LIN {X 0,Y 87.891,Z 1219.976,A -85,B 0,C 180,E1 32199.229,E2 32199.229} C_VEL
LIN {X 0,Y 83.761,Z 1226.847,A -85,B 0,C 180,E1 32206.195,E2 32206.195} C_VEL
LIN {X 0,Y 77.904,Z 1236.707,A -85,B 0,C 180,E1 32219.704,E2 32219.704} C_VEL
LIN {X 0,Y 80.765,Z 1249.005,A -85,B 0,C 180,E1 32238.354,E2 32238.354} C_VEL
LIN {X 0,Y 97.105,Z 1263.122,A -85,B 0,C 180,E1 32262.701,E2 32262.701} C_VEL
LIN {X 0,Y 95.268,Z 1262.7,A -85,B 0,C 180,E1 32265.572,E2 32265.572} C_VEL
LIN {X 0,Y 81.258,Z 1251.243,A -85,B 0,C 180,E1 32296.572,E2 32296.572} C_VEL
LIN {X 0,Y 81.376,Z 1245.78,A -85,B 0,C 180,E1 32307.381,E2 32307.381} C_VEL
LIN {X 0,Y 84.468,Z 1224.374,A -85,B 0,C 180,E1 32333.558,E2 32333.558} C_VEL
LIN {X 0,Y 99.54,Z 1230.344,A -85,B 0,C 180,E1 32359.626,E2 32359.626} C_VEL
LIN {X 0,Y 109.101,Z 1231.557,A -85,B 0,C 180,E1 32366.508,E2 32366.508} C_VEL
LIN {X 0,Y 89.421,Z 1216.791,A -85,B 0,C 180,E1 32382.617,E2 32382.617} C_VEL
LIN {X 0,Y 79.635,Z 1196.68,A -85,B 0,C 180,E1 32404.169,E2 32404.169} C_VEL
LIN {X 0,Y 80.434,Z 1173.933,A -85,B 0,C 180,E1 32423.679,E2 32423.679} C_VEL
LIN {X 0,Y 87.564,Z 1144.411,A -85,B 0,C 180,E1 32440.462,E2 32440.462} C_VEL
LIN {X 0,Y 96.99,Z 1111.48,A -85,B 0,C 180,E1 32451.459,E2 32451.459} C_VEL
LIN {X 0,Y 103.746,Z 1084.246,A -85,B 0,C 180,E1 32457.336,E2 32457.336} C_VEL
LIN {X 0,Y 98.146,Z 1049.051,A -85,B 0,C 180,E1 32468.442,E2 32468.442} C_VEL
LIN {X 0,Y 97.255,Z 1043.42,A -85,B 0,C 180,E1 32470.62,E2 32470.62} C_VEL
LIN {X 0,Y 108.101,Z 1031.914,A -85,B 0,C 180,E1 32479.137,E2 32479.137} C_VEL
LIN {X 0,Y 113.422,Z 1053.158,A -85,B 0,C 180,E1 32489.964,E2 32489.964} C_VEL
LIN {X 0,Y 118.845,Z 1081.531,A -85,B 0,C 180,E1 32501.191,E2 32501.191} C_VEL
LIN {X 0,Y 122.921,Z 1111.426,A -85,B 0,C 180,E1 32511.669,E2 32511.669} C_VEL
LIN {X 0,Y 123.967,Z 1124.968,A -85,B 0,C 180,E1 32516.233,E2 32516.233} C_VEL
LIN {X 0,Y 105.518,Z 1162.751,A -85,B 0,C 180,E1 32526.032,E2 32526.032} C_VEL
LIN {X 0,Y 89.617,Z 1194.356,A -85,B 0,C 180,E1 32540.566,E2 32540.566} C_VEL
LIN {X 0,Y 79.544,Z 1220.884,A -85,B 0,C 180,E1 32561.434,E2 32561.434} C_VEL
LIN {X 0,Y 77.904,Z 1236.707,A -85,B 0,C 180,E1 32579.704,E2 32579.704} C_VEL
LIN {X 0,Y 76.332,Z 1241.977,A -85,B 0,C 180,E1 32588.571,E2 32588.571} C_VEL
LIN {X 0,Y 75.282,Z 1248.971,A -85,B 0,C 180,E1 32604.581,E2 32604.581} C_VEL
LIN {X 0,Y 88.436,Z 1259.457,A -85,B 0,C 180,E1 32623.162,E2 32623.162} C_VEL
LIN {X 0,Y 74.447,Z 1249.413,A -85,B 0,C 180,E1 32652.297,E2 32652.297} C_VEL
LIN {X 0,Y 73.972,Z 1242.557,A -85,B 0,C 180,E1 32667.119,E2 32667.119} C_VEL
LIN {X 0,Y 77.694,Z 1220.967,A -85,B 0,C 180,E1 32695.202,E2 32695.202} C_VEL
LIN {X 0,Y 96.727,Z 1227.821,A -85,B 0,C 180,E1 32724.628,E2 32724.628} C_VEL
LIN {X 0,Y 98.246,Z 1227.61,A -85,B 0,C 180,E1 32726.965,E2 32726.965} C_VEL
LIN {X 0,Y 77.889,Z 1209.389,A -85,B 0,C 180,E1 32746.807,E2 32746.807} C_VEL
LIN {X 0,Y 71.41,Z 1187.367,A -85,B 0,C 180,E1 32770.787,E2 32770.787} C_VEL
LIN {X 0,Y 74.839,Z 1162.016,A -85,B 0,C 180,E1 32791.346,E2 32791.346} C_VEL
LIN {X 0,Y 83.559,Z 1131.844,A -85,B 0,C 180,E1 32806.599,E2 32806.599} C_VEL
LIN {X 0,Y 93.999,Z 1095.283,A -85,B 0,C 180,E1 32816.978,E2 32816.978} C_VEL
LIN {X 0,Y 96.451,Z 1084.975,A -85,B 0,C 180,E1 32819.249,E2 32819.249} C_VEL
LIN {X 0,Y 92.458,Z 1055.079,A -85,B 0,C 180,E1 32829.571,E2 32829.571} C_VEL
LIN {X 0,Y 102.072,Z 1044.415,A -85,B 0,C 180,E1 32837.324,E2 32837.324} C_VEL
LIN {X 0,Y 105.365,Z 1042.471,A -85,B 0,C 180,E1 32840.02,E2 32840.02} C_VEL
LIN {X 0,Y 109.77,Z 1064.935,A -85,B 0,C 180,E1 32851.137,E2 32851.137} C_VEL
LIN {X 0,Y 114.019,Z 1094.414,A -85,B 0,C 180,E1 32862.923,E2 32862.923} C_VEL
LIN {X 0,Y 116.99,Z 1124.374,A -85,B 0,C 180,E1 32873.982,E2 32873.982} C_VEL
LIN {X 0,Y 100.249,Z 1158.488,A -85,B 0,C 180,E1 32882.924,E2 32882.924} C_VEL
LIN {X 0,Y 83.092,Z 1191.044,A -85,B 0,C 180,E1 32897.939,E2 32897.939} C_VEL
LIN {X 0,Y 72.698,Z 1215.97,A -85,B 0,C 180,E1 32918.055,E2 32918.055} C_VEL
LIN {X 0,Y 70.433,Z 1234.644,A -85,B 0,C 180,E1 32940.852,E2 32940.852} C_VEL
LIN {X 0,Y 73.816,Z 1246.719,A -85,B 0,C 180,E1 32960.556,E2 32960.556} C_VEL
LIN {X 0,Y 75.282,Z 1248.971,A -85,B 0,C 180,E1 32964.581,E2 32964.581} C_VEL
LIN {X 0,Y 75.8,Z 1251.791,A -85,B 0,C 180,E1 32973.282,E2 32973.282} C_VEL
LIN {X 0,Y 77.991,Z 1254.326,A -85,B 0,C 180,E1 32981.785,E2 32981.785} C_VEL
LIN {X 0,Y 79.566,Z 1255.315,A -85,B 0,C 180,E1 32983.483,E2 32983.483} C_VEL
LIN {X 0,Y 67.204,Z 1245.094,A -85,B 0,C 180,E1 33013.693,E2 33013.693} C_VEL
LIN {X 0,Y 66.603,Z 1239.116,A -85,B 0,C 180,E1 33026.8,E2 33026.8} C_VEL
LIN {X 0,Y 70.218,Z 1218.237,A -85,B 0,C 180,E1 33055.632,E2 33055.632} C_VEL
LIN {X 0,Y 71.218,Z 1217.611,A -85,B 0,C 180,E1 33058.093,E2 33058.093} C_VEL
LIN {X 0,Y 85.672,Z 1223.54,A -85,B 0,C 180,E1 33082.924,E2 33082.924} C_VEL
LIN {X 0,Y 88.018,Z 1223.499,A -85,B 0,C 180,E1 33086.565,E2 33086.565} C_VEL
LIN {X 0,Y 68.507,Z 1203.689,A -85,B 0,C 180,E1 33108.934,E2 33108.934} C_VEL
LIN {X 0,Y 63.835,Z 1180.307,A -85,B 0,C 180,E1 33135.353,E2 33135.353} C_VEL
LIN {X 0,Y 69.107,Z 1153.051,A -85,B 0,C 180,E1 33157.19,E2 33157.19} C_VEL
LIN {X 0,Y 79.014,Z 1121.692,A -85,B 0,C 180,E1 33171.823,E2 33171.823} C_VEL
LIN {X 0,Y 89.139,Z 1085.188,A -85,B 0,C 180,E1 33181.58,E2 33181.58} C_VEL
LIN {X 0,Y 87.192,Z 1066.85,A -85,B 0,C 180,E1 33188.4,E2 33188.4} C_VEL
LIN {X 0,Y 100.232,Z 1053.075,A -85,B 0,C 180,E1 33198.848,E2 33198.848} C_VEL
LIN {X 0,Y 101.967,Z 1052.089,A -85,B 0,C 180,E1 33200.229,E2 33200.229} C_VEL
LIN {X 0,Y 105.404,Z 1075.537,A -85,B 0,C 180,E1 33211.796,E2 33211.796} C_VEL
LIN {X 0,Y 108.342,Z 1104.004,A -85,B 0,C 180,E1 33223.613,E2 33223.613} C_VEL
LIN {X 0,Y 109.485,Z 1126.882,A -85,B 0,C 180,E1 33232.443,E2 33232.443} C_VEL
LIN {X 0,Y 89.571,Z 1164.561,A -85,B 0,C 180,E1 33243.24,E2 33243.24} C_VEL
LIN {X 0,Y 72.3,Z 1196.33,A -85,B 0,C 180,E1 33260.938,E2 33260.938} C_VEL
LIN {X 0,Y 63.495,Z 1221.244,A -85,B 0,C 180,E1 33286.095,E2 33286.095} C_VEL
LIN {X 0,Y 63.969,Z 1237.279,A -85,B 0,C 180,E1 33310.134,E2 33310.134} C_VEL
LIN {X 0,Y 76.453,Z 1253.317,A -85,B 0,C 180,E1 33339.989,E2 33339.989} C_VEL
LIN {X 0,Y 77.991,Z 1254.326,A -85,B 0,C 180,E1 33341.785,E2 33341.785} C_VEL
LIN {X 0,Y 77.258,Z 1254.281,A -85,B 0,C 180,E1 33345.005,E2 33345.005} C_VEL
LIN {X 0,Y 64.108,Z 1246.977,A -85,B 0,C 180,E1 33356.202,E2 33356.202} C_VEL
LIN {X 0,Y 59.76,Z 1237.461,A -85,B 0,C 180,E1 33382.785,E2 33382.785} C_VEL
LIN {X 0,Y 63.054,Z 1215.304,A -85,B 0,C 180,E1 33416.853,E2 33416.853} C_VEL
LIN {X 0,Y 64.644,Z 1213.641,A -85,B 0,C 180,E1 33419.626,E2 33419.626} C_VEL
LIN {X 0,Y 79.165,Z 1219.797,A -85,B 0,C 180,E1 33445.055,E2 33445.055} C_VEL
LIN {X 0,Y 60.185,Z 1199.211,A -85,B 0,C 180,E1 33469.222,E2 33469.222} C_VEL
LIN {X 0,Y 56.306,Z 1176.169,A -85,B 0,C 180,E1 33497.193,E2 33497.193} C_VEL
LIN {X 0,Y 62.593,Z 1148.344,A -85,B 0,C 180,E1 33520.711,E2 33520.711} C_VEL
LIN {X 0,Y 73.042,Z 1116.882,A -85,B 0,C 180,E1 33535.493,E2 33535.493} C_VEL
LIN {X 0,Y 82.106,Z 1086.586,A -85,B 0,C 180,E1 33543.861,E2 33543.861} C_VEL
LIN {X 0,Y 81.443,Z 1078.77,A -85,B 0,C 180,E1 33547.041,E2 33547.041} C_VEL
LIN {X 0,Y 90.144,Z 1069.603,A -85,B 0,C 180,E1 33554.948,E2 33554.948} C_VEL
LIN {X 0,Y 98.19,Z 1061.545,A -85,B 0,C 180,E1 33560.336,E2 33560.336} C_VEL
LIN {X 0,Y 100.592,Z 1086.487,A -85,B 0,C 180,E1 33572.658,E2 33572.658} C_VEL
LIN {X 0,Y 102.49,Z 1116.067,A -85,B 0,C 180,E1 33585.503,E2 33585.503} C_VEL
LIN {X 0,Y 102.577,Z 1127.464,A -85,B 0,C 180,E1 33590.14,E2 33590.14} C_VEL
LIN {X 0,Y 82.03,Z 1164.658,A -85,B 0,C 180,E1 33601.179,E2 33601.179} C_VEL
LIN {X 0,Y 63.691,Z 1197.177,A -85,B 0,C 180,E1 33621.235,E2 33621.235} C_VEL
LIN {X 0,Y 55.517,Z 1221.624,A -85,B 0,C 180,E1 33650.066,E2 33650.066} C_VEL
LIN {X 0,Y 57.383,Z 1236.242,A -85,B 0,C 180,E1 33675.197,E2 33675.197} C_VEL
LIN {X 0,Y 70.051,Z 1250.327,A -85,B 0,C 180,E1 33702.903,E2 33702.903} C_VEL
LIN {X 0,Y 69.694,Z 1250.337,A -85,B 0,C 180,E1 33705.879,E2 33705.879} C_VEL
LIN {X 0,Y 64.108,Z 1246.977,A -85,B 0,C 180,E1 33716.202,E2 33716.202} C_VEL
LIN {X 0,Y 59.041,Z 1242.349,A -85,B 0,C 180,E1 33726.703,E2 33726.703} C_VEL
LIN {X 0,Y 51.942,Z 1231.806,A -85,B 0,C 180,E1 33745.881,E2 33745.881} C_VEL
LIN {X 0,Y 55.921,Z 1212.323,A -85,B 0,C 180,E1 33778.388,E2 33778.388} C_VEL
LIN {X 0,Y 58.466,Z 1209.764,A -85,B 0,C 180,E1 33782.484,E2 33782.484} C_VEL
LIN {X 0,Y 69.398,Z 1214.751,A -85,B 0,C 180,E1 33804.234,E2 33804.234} C_VEL
LIN {X 0,Y 51.296,Z 1192.908,A -85,B 0,C 180,E1 33831.63,E2 33831.63} C_VEL
LIN {X 0,Y 49.21,Z 1169.418,A -85,B 0,C 180,E1 33862.305,E2 33862.305} C_VEL
LIN {X 0,Y 57.231,Z 1140.499,A -85,B 0,C 180,E1 33886.802,E2 33886.802} C_VEL
LIN {X 0,Y 68.471,Z 1108.56,A -85,B 0,C 180,E1 33900.791,E2 33900.791} C_VEL
LIN {X 0,Y 73.618,Z 1093.919,A -85,B 0,C 180,E1 33905.231,E2 33905.231} C_VEL
LIN {X 0,Y 80.38,Z 1085.165,A -85,B 0,C 180,E1 33910.698,E2 33910.698} C_VEL
LIN {X 0,Y 94.02,Z 1071.635,A -85,B 0,C 180,E1 33920.682,E2 33920.682} C_VEL
LIN {X 0,Y 95.375,Z 1097.988,A -85,B 0,C 180,E1 33933.943,E2 33933.943} C_VEL
LIN {X 0,Y 96.076,Z 1126.611,A -85,B 0,C 180,E1 33947.037,E2 33947.037} C_VEL
LIN {X 0,Y 77.545,Z 1159.832,A -85,B 0,C 180,E1 33956.77,E2 33956.77} C_VEL
LIN {X 0,Y 58.907,Z 1190.664,A -85,B 0,C 180,E1 33974.835,E2 33974.835} C_VEL
LIN {X 0,Y 48.611,Z 1215.176,A -85,B 0,C 180,E1 34004.042,E2 34004.042} C_VEL
LIN {X 0,Y 49.501,Z 1231.116,A -85,B 0,C 180,E1 34033.142,E2 34033.142} C_VEL
LIN {X 0,Y 60.95,Z 1245.145,A -85,B 0,C 180,E1 34062.662,E2 34062.662} C_VEL
LIN {X 0,Y 62.147,Z 1245.993,A -85,B 0,C 180,E1 34064.925,E2 34064.925} C_VEL
LIN {X 0,Y 52.986,Z 1235.578,A -85,B 0,C 180,E1 34097.693,E2 34097.693} C_VEL
LIN {X 0,Y 51.942,Z 1231.806,A -85,B 0,C 180,E1 34105.881,E2 34105.881} C_VEL
LIN {X 0,Y 48.765,Z 1226.669,A -85,B 0,C 180,E1 34113.21,E2 34113.21} C_VEL
LIN {X 0,Y 44.181,Z 1218.19,A -85,B 0,C 180,E1 34124.906,E2 34124.906} C_VEL
LIN {X 0,Y 44.33,Z 1217.33,A -85,B 0,C 180,E1 34126.466,E2 34126.466} C_VEL
LIN {X 0,Y 52.377,Z 1205.621,A -85,B 0,C 180,E1 34145.447,E2 34145.447} C_VEL
LIN {X 0,Y 59.691,Z 1209.1,A -85,B 0,C 180,E1 34163.091,E2 34163.091} C_VEL
LIN {X 0,Y 42.559,Z 1185.93,A -85,B 0,C 180,E1 34195.04,E2 34195.04} C_VEL
LIN {X 0,Y 42.869,Z 1160.631,A -85,B 0,C 180,E1 34230.558,E2 34230.558} C_VEL
LIN {X 0,Y 53.258,Z 1130.529,A -85,B 0,C 180,E1 34254.746,E2 34254.746} C_VEL
LIN {X 0,Y 57.065,Z 1121.956,A -85,B 0,C 180,E1 34259.856,E2 34259.856} C_VEL
LIN {X 0,Y 67.287,Z 1108.028,A -85,B 0,C 180,E1 34267.679,E2 34267.679} C_VEL
LIN {X 0,Y 75.787,Z 1095.542,A -85,B 0,C 180,E1 34271.676,E2 34271.676} C_VEL
LIN {X 0,Y 87.589,Z 1083.735,A -85,B 0,C 180,E1 34279.991,E2 34279.991} C_VEL
LIN {X 0,Y 89.518,Z 1083.35,A -85,B 0,C 180,E1 34281.942,E2 34281.942} C_VEL
LIN {X 0,Y 89.573,Z 1110.852,A -85,B 0,C 180,E1 34296.024,E2 34296.024} C_VEL
LIN {X 0,Y 88.791,Z 1129.288,A -85,B 0,C 180,E1 34304.791,E2 34304.791} C_VEL
LIN {X 0,Y 66.705,Z 1165.596,A -85,B 0,C 180,E1 34316.287,E2 34316.287} C_VEL
LIN {X 0,Y 47.315,Z 1196.779,A -85,B 0,C 180,E1 34340.005,E2 34340.005} C_VEL
LIN {X 0,Y 40.646,Z 1220.731,A -85,B 0,C 180,E1 34379.848,E2 34379.848} C_VEL
LIN {X 0,Y 46.018,Z 1233.755,A -85,B 0,C 180,E1 34409.44,E2 34409.44} C_VEL
LIN {X 0,Y 53.265,Z 1240.453,A -85,B 0,C 180,E1 34424.393,E2 34424.393} C_VEL
LIN {X 0,Y 47.097,Z 1234.827,A -85,B 0,C 180,E1 34446.38,E2 34446.38} C_VEL
LIN {X 0,Y 45.103,Z 1229.131,A -85,B 0,C 180,E1 34462.47,E2 34462.47} C_VEL
LIN {X 0,Y 44.33,Z 1217.33,A -85,B 0,C 180,E1 34486.466,E2 34486.466} C_VEL
LIN {X 0,Y 45.397,Z 1202.633,A -85,B 0,C 180,E1 34508.049,E2 34508.049} C_VEL
LIN {X 0,Y 46.237,Z 1201.824,A -85,B 0,C 180,E1 34509.167,E2 34509.167} C_VEL
LIN {X 0,Y 50.521,Z 1203.175,A -85,B 0,C 180,E1 34521.115,E2 34521.115} C_VEL
LIN {X 0,Y 34.096,Z 1178.233,A -85,B 0,C 180,E1 34560.182,E2 34560.182} C_VEL
LIN {X 0,Y 38.126,Z 1150.199,A -85,B 0,C 180,E1 34603.499,E2 34603.499} C_VEL
LIN {X 0,Y 49.75,Z 1134.636,A -85,B 0,C 180,E1 34621.608,E2 34621.608} C_VEL
LIN {X 0,Y 59.021,Z 1123.149,A -85,B 0,C 180,E1 34628.808,E2 34628.808} C_VEL
LIN {X 0,Y 72.062,Z 1105.931,A -85,B 0,C 180,E1 34634.921,E2 34634.921} C_VEL
LIN {X 0,Y 77.731,Z 1098.677,A -85,B 0,C 180,E1 34637.411,E2 34637.411} C_VEL
LIN {X 0,Y 84.478,Z 1092.587,A -85,B 0,C 180,E1 34641.733,E2 34641.733} C_VEL
LIN {X 0,Y 83.245,Z 1119.949,A -85,B 0,C 180,E1 34656.484,E2 34656.484} C_VEL
LIN {X 0,Y 82.377,Z 1129.72,A -85,B 0,C 180,E1 34661.404,E2 34661.404} C_VEL
LIN {X 0,Y 59.468,Z 1165.644,A -85,B 0,C 180,E1 34672.822,E2 34672.822} C_VEL
LIN {X 0,Y 39.115,Z 1196.45,A -85,B 0,C 180,E1 34699.109,E2 34699.109} C_VEL
LIN {X 0,Y 33.742,Z 1219.483,A -85,B 0,C 180,E1 34746.261,E2 34746.261} C_VEL
LIN {X 0,Y 41.786,Z 1232.339,A -85,B 0,C 180,E1 34779.193,E2 34779.193} C_VEL
LIN {X 0,Y 44.847,Z 1234.9,A -85,B 0,C 180,E1 34787.609,E2 34787.609} C_VEL
LIN {X 0,Y 38.885,Z 1227.151,A -85,B 0,C 180,E1 34816.011,E2 34816.011} C_VEL
LIN {X 0,Y 41.984,Z 1205.954,A -85,B 0,C 180,E1 34862.891,E2 34862.891} C_VEL
LIN {X 0,Y 46.237,Z 1201.824,A -85,B 0,C 180,E1 34869.167,E2 34869.167} C_VEL
LIN {X 0,Y 45.472,Z 1200.157,A -85,B 0,C 180,E1 34874.838,E2 34874.838} C_VEL
LIN {X 0,Y 38.074,Z 1193.408,A -85,B 0,C 180,E1 34883.882,E2 34883.882} C_VEL
LIN {X 0,Y 33.671,Z 1188.156,A -85,B 0,C 180,E1 34890.682,E2 34890.682} C_VEL
LIN {X 0,Y 30.735,Z 1160.605,A -85,B 0,C 180,E1 34962.948,E2 34962.948} C_VEL
LIN {X 0,Y 49.686,Z 1138.105,A -85,B 0,C 180,E1 34989.762,E2 34989.762} C_VEL
LIN {X 0,Y 69.499,Z 1115.098,A -85,B 0,C 180,E1 34999.407,E2 34999.407} C_VEL
LIN {X 0,Y 76.781,Z 1105.196,A -85,B 0,C 180,E1 35001.126,E2 35001.126} C_VEL
LIN {X 0,Y 78.878,Z 1104.044,A -85,B 0,C 180,E1 35002.788,E2 35002.788} C_VEL
LIN {X 0,Y 76.499,Z 1129.664,A -85,B 0,C 180,E1 35017.395,E2 35017.395} C_VEL
LIN {X 0,Y 51.301,Z 1167.335,A -85,B 0,C 180,E1 35029.342,E2 35029.342} C_VEL
LIN {X 0,Y 29.382,Z 1198.835,A -85,B 0,C 180,E1 35063.175,E2 35063.175} C_VEL
LIN {X 0,Y 27.431,Z 1218.111,A -85,B 0,C 180,E1 35115.796,E2 35115.796} C_VEL
LIN {X 0,Y 36.783,Z 1229.079,A -85,B 0,C 180,E1 35146.728,E2 35146.728} C_VEL
LIN {X 0,Y 33.645,Z 1225.762,A -85,B 0,C 180,E1 35163.82,E2 35163.82} C_VEL
LIN {X 0,Y 29.359,Z 1216.926,A -85,B 0,C 180,E1 35190.137,E2 35190.137} C_VEL
LIN {X 0,Y 37.806,Z 1200.14,A -85,B 0,C 180,E1 35230.78,E2 35230.78} C_VEL
LIN {X 0,Y 42.029,Z 1197.257,A -85,B 0,C 180,E1 35236.28,E2 35236.28} C_VEL
LIN {X 0,Y 33.671,Z 1188.156,A -85,B 0,C 180,E1 35250.682,E2 35250.682} C_VEL
LIN {X 0,Y 27.603,Z 1184.456,A -85,B 0,C 180,E1 35260.544,E2 35260.544} C_VEL
LIN {X 0,Y 19.659,Z 1180.506,A -85,B 0,C 180,E1 35285.817,E2 35285.817} C_VEL
LIN {X 0,Y 19.527,Z 1179.715,A -85,B 0,C 180,E1 35289.487,E2 35289.487} C_VEL
LIN {X 0,Y 38.387,Z 1153.882,A -85,B 0,C 180,E1 35350.084,E2 35350.084} C_VEL
LIN {X 0,Y 71.222,Z 1118.891,A -85,B 0,C 180,E1 35364.913,E2 35364.913} C_VEL
LIN {X 0,Y 72.192,Z 1119.094,A -85,B 0,C 180,E1 35366.166,E2 35366.166} C_VEL
LIN {X 0,Y 70.432,Z 1130.498,A -85,B 0,C 180,E1 35373.005,E2 35373.005} C_VEL
LIN {X 0,Y 44.055,Z 1167.961,A -85,B 0,C 180,E1 35384.144,E2 35384.144} C_VEL
LIN {X 0,Y 21.39,Z 1197.787,A -85,B 0,C 180,E1 35421.331,E2 35421.331} C_VEL
LIN {X 0,Y 22.315,Z 1216.643,A -85,B 0,C 180,E1 35490.289,E2 35490.289} C_VEL
LIN {X 0,Y 28.739,Z 1222.889,A -85,B 0,C 180,E1 35509.286,E2 35509.286} C_VEL
LIN {X 0,Y 26.873,Z 1220.739,A -85,B 0,C 180,E1 35521.484,E2 35521.484} C_VEL
LIN {X 0,Y 28.608,Z 1199.305,A -85,B 0,C 180,E1 35591.27,E2 35591.27} C_VEL
LIN {X 0,Y 31.073,Z 1197.019,A -85,B 0,C 180,E1 35595.57,E2 35595.57} C_VEL
LIN {X 0,Y 28.116,Z 1192.896,A -85,B 0,C 180,E1 35603.668,E2 35603.668} C_VEL
LIN {X 0,Y 19.527,Z 1179.715,A -85,B 0,C 180,E1 35649.487,E2 35649.487} C_VEL
LIN {X 0,Y 22.626,Z 1171.188,A -85,B 0,C 180,E1 35690.944,E2 35690.944} C_VEL
LIN {X 0,Y 32.782,Z 1162.726,A -85,B 0,C 180,E1 35715.399,E2 35715.399} C_VEL
LIN {X 0,Y 51.213,Z 1146.029,A -85,B 0,C 180,E1 35725.295,E2 35725.295} C_VEL
LIN {X 0,Y 60.763,Z 1136.3,A -85,B 0,C 180,E1 35727.645,E2 35727.645} C_VEL
LIN {X 0,Y 59.697,Z 1138.88,A -85,B 0,C 180,E1 35728.943,E2 35728.943} C_VEL
LIN {X 0,Y 32.775,Z 1173.667,A -85,B 0,C 180,E1 35739.724,E2 35739.724} C_VEL
LIN {X 0,Y 11.428,Z 1201.008,A -85,B 0,C 180,E1 35800.067,E2 35800.067} C_VEL
LIN {X 0,Y 19.336,Z 1215.022,A -85,B 0,C 180,E1 35871.076,E2 35871.076} C_VEL
LIN {X 0,Y 17.097,Z 1212.134,A -85,B 0,C 180,E1 35887.496,E2 35887.496} C_VEL
LIN {X 0,Y 21.143,Z 1196.952,A -85,B 0,C 180,E1 35956.055,E2 35956.055} C_VEL
LIN {X 0,Y 15.22,Z 1190.048,A -85,B 0,C 180,E1 35981.645,E2 35981.645} C_VEL
LIN {X 0,Y 26.63,Z 1168.462,A -85,B 0,C 180,E1 36069.373,E2 36069.373} C_VEL
LIN {X 0,Y 32.782,Z 1162.726,A -85,B 0,C 180,E1 36075.399,E2 36075.399} C_VEL
LIN {X 0,Y 32.232,Z 1165.337,A -85,B 0,C 180,E1 36080.699,E2 36080.699} C_VEL
LIN {X 0,Y 22.619,Z 1178.129,A -85,B 0,C 180,E1 36089.734,E2 36089.734} C_VEL
LIN {X 0,Y 19.771,Z 1181.155,A -85,B 0,C 180,E1 36091.79,E2 36091.79} C_VEL
LIN {X 0,Y 8.559,Z 1205.113,A -85,B 0,C 180,E1 36236.286,E2 36236.286} C_VEL
LIN {X 0,Y 8.113,Z 1202.65,A -85,B 0,C 180,E1 36270.497,E2 36270.497} C_VEL
LIN {X 0,Y 10.568,Z 1197.619,A -85,B 0,C 180,E1 36312.666,E2 36312.666} C_VEL
LIN {X 0,Y 10.601,Z 1195.82,A -85,B 0,C 180,E1 36321.939,E2 36321.939} C_VEL
LIN {X 0,Y 24.976,Z 1173.819,A -85,B 0,C 180,E1 36443.208,E2 36443.208} C_VEL
LIN {X 0,Y 30.497,Z 1169.161,A -85,B 0,C 180,E1 36445.659,E2 36445.659} C_VEL
LIN {X 0,Y 19.771,Z 1181.155,A -85,B 0,C 180,E1 36451.79,E2 36451.79} C_VEL
LIN {X 0,Y 19.193,Z 1182.578,A -85,B 0,C 180,E1 36452.194,E2 36452.194} C_VEL
LIN {X 0,Y 19.193,Z 1317.5,A -85,B 0,C 180,E1 36452.194,E2 36452.194} C_VEL
LIN {X 0,Y 19.193,Z 1317.5,A -85,B 0,C 180,E1 36452.194,E2 36452.194}

QRS_NEXT_CUT()
PTP {E1 36537.214,E2 36537.214}
PTP {X 0,Y 759.913,A -85,B 0,C 180,E1 36537.214,E2 36537.214,E3 0,E4 0,E5 0,E6 0}
QRS_SPEED_INIT()
LIN {X 0,Y 759.913,Z 1317.5,A -85,B 0,C 180,E1 36537.214,E2 36537.214,E3 0,E4 0,E5 0,E6 0} C_VEL
LIN {X 0,Y 759.913,Z 1255.248,A -85,B 0,C 180,E1 36537.214,E2 36537.214} C_VEL
LIN {X 0,Y 759.913,Z 1246.975,A -85,B 0,C 180,E1 36537.214,E2 36537.214} C_VEL
LIN {X 0,Y 759.904,Z 1244.988,A -85,B 0,C 180,E1 36537.08,E2 36537.08} C_VEL
LIN {X 0,Y 759.916,Z 1241.315,A -85,B 0,C 180,E1 36535.472,E2 36535.472} C_VEL
LIN {X 0,Y 759.911,Z 1235.849,A -85,B 0,C 180,E1 36533.806,E2 36533.806} C_VEL
LIN {X 0,Y 759.916,Z 1228.905,A -85,B 0,C 180,E1 36532.211,E2 36532.211} C_VEL
LIN {X 0,Y 759.9,Z 1220.481,A -85,B 0,C 180,E1 36530.686,E2 36530.686} C_VEL
LIN {X 0,Y 759.915,Z 1210.302,A -85,B 0,C 180,E1 36529.155,E2 36529.155} C_VEL
LIN {X 0,Y 759.906,Z 1198.713,A -85,B 0,C 180,E1 36527.692,E2 36527.692} C_VEL
LIN {X 0,Y 759.909,Z 1185.675,A -85,B 0,C 180,E1 36526.3,E2 36526.3} C_VEL
LIN {X 0,Y 759.917,Z 1170.403,A -85,B 0,C 180,E1 36524.899,E2 36524.899} C_VEL
LIN {X 0,Y 759.911,Z 1154.515,A -85,B 0,C 180,E1 36523.645,E2 36523.645} C_VEL
LIN {X 0,Y 759.916,Z 1137.114,A -85,B 0,C 180,E1 36522.463,E2 36522.463} C_VEL
LIN {X 0,Y 759.916,Z 1119.277,A -85,B 0,C 180,E1 36521.432,E2 36521.432} C_VEL
LIN {X 0,Y 759.918,Z 1099.934,A -85,B 0,C 180,E1 36520.475,E2 36520.475} C_VEL
LIN {X 0,Y 759.918,Z 1080.841,A -85,B 0,C 180,E1 36519.673,E2 36519.673} C_VEL
LIN {X 0,Y 759.913,Z 1060.872,A -85,B 0,C 180,E1 36518.988,E2 36518.988} C_VEL
LIN {X 0,Y 759.912,Z 1038.847,A -85,B 0,C 180,E1 36518.381,E2 36518.381} C_VEL
LIN {X 0,Y 759.907,Z 1017.58,A -85,B 0,C 180,E1 36517.935,E2 36517.935} C_VEL
LIN {X 0,Y 759.914,Z 996.129,A -85,B 0,C 180,E1 36517.629,E2 36517.629} C_VEL
LIN {X 0,Y 759.91,Z 700.151,A -85,B 0,C 180,E1 36514.625,E2 36514.625} C_VEL
LIN {X 0,Y 759.888,Z 662.004,A -85,B 0,C 180,E1 36511.811,E2 36511.811} C_VEL
LIN {X 0,Y 759.891,Z 638.011,A -85,B 0,C 180,E1 36509.977,E2 36509.977} C_VEL
LIN {X 0,Y 759.905,Z 638.009,A -85,B 0,C 180,E1 36507.082,E2 36507.082} C_VEL
LIN {X 0,Y 759.905,Z 638.01,A -85,B 0,C 180,E1 36504.252,E2 36504.252} C_VEL
LIN {X 0,Y 759.89,Z 638.008,A -85,B 0,C 180,E1 36501.408,E2 36501.408} C_VEL
LIN {X 0,Y 759.918,Z 638.015,A -85,B 0,C 180,E1 36498.559,E2 36498.559} C_VEL
LIN {X 0,Y 759.908,Z 638.006,A -85,B 0,C 180,E1 36495.601,E2 36495.601} C_VEL
LIN {X 0,Y 759.907,Z 638.006,A -85,B 0,C 180,E1 36492.647,E2 36492.647} C_VEL
LIN {X 0,Y 759.902,Z 638.015,A -85,B 0,C 180,E1 36489.754,E2 36489.754} C_VEL
LIN {X 0,Y 759.889,Z 638.007,A -85,B 0,C 180,E1 36486.966,E2 36486.966} C_VEL
LIN {X 0,Y 759.903,Z 638.013,A -85,B 0,C 180,E1 36484.142,E2 36484.142} C_VEL
LIN {X 0,Y 759.907,Z 638.007,A -85,B 0,C 180,E1 36481.316,E2 36481.316} C_VEL
LIN {X 0,Y 759.892,Z 638.009,A -85,B 0,C 180,E1 36478.447,E2 36478.447} C_VEL
LIN {X 0,Y 759.894,Z 638.013,A -85,B 0,C 180,E1 36475.664,E2 36475.664} C_VEL
LIN {X 0,Y 759.914,Z 638.004,A -85,B 0,C 180,E1 36472.841,E2 36472.841} C_VEL
LIN {X 0,Y 759.919,Z 638.008,A -85,B 0,C 180,E1 36469.765,E2 36469.765} C_VEL
LIN {X 0,Y 759.896,Z 638.01,A -85,B 0,C 180,E1 36466.906,E2 36466.906} C_VEL
LIN {X 0,Y 759.889,Z 638.008,A -85,B 0,C 180,E1 36464.09,E2 36464.09} C_VEL
LIN {X 0,Y 759.905,Z 638.013,A -85,B 0,C 180,E1 36461.307,E2 36461.307} C_VEL
LIN {X 0,Y 759.913,Z 638.004,A -85,B 0,C 180,E1 36458.317,E2 36458.317} C_VEL
LIN {X 0,Y 759.911,Z 638.006,A -85,B 0,C 180,E1 36455.286,E2 36455.286} C_VEL
LIN {X 0,Y 759.905,Z 638.015,A -85,B 0,C 180,E1 36452.339,E2 36452.339} C_VEL
LIN {X 0,Y 759.889,Z 638.007,A -85,B 0,C 180,E1 36449.549,E2 36449.549} C_VEL
LIN {X 0,Y 759.907,Z 638.013,A -85,B 0,C 180,E1 36446.758,E2 36446.758} C_VEL
LIN {X 0,Y 759.907,Z 638.007,A -85,B 0,C 180,E1 36443.883,E2 36443.883} C_VEL
LIN {X 0,Y 759.892,Z 638.008,A -85,B 0,C 180,E1 36440.993,E2 36440.993} C_VEL
LIN {X 0,Y 759.893,Z 638.013,A -85,B 0,C 180,E1 36438.232,E2 36438.232} C_VEL
LIN {X 0,Y 759.91,Z 638.005,A -85,B 0,C 180,E1 36435.368,E2 36435.368} C_VEL
LIN {X 0,Y 759.916,Z 638.008,A -85,B 0,C 180,E1 36432.307,E2 36432.307} C_VEL
LIN {X 0,Y 759.897,Z 638.011,A -85,B 0,C 180,E1 36429.433,E2 36429.433} C_VEL
LIN {X 0,Y 759.888,Z 638.008,A -85,B 0,C 180,E1 36426.587,E2 36426.587} C_VEL
LIN {X 0,Y 759.912,Z 638.015,A -85,B 0,C 180,E1 36423.763,E2 36423.763} C_VEL
LIN {X 0,Y 759.915,Z 638.005,A -85,B 0,C 180,E1 36420.868,E2 36420.868} C_VEL
LIN {X 0,Y 759.914,Z 638.005,A -85,B 0,C 180,E1 36417.8,E2 36417.8} C_VEL
LIN {X 0,Y 759.919,Z 638.014,A -85,B 0,C 180,E1 36414.796,E2 36414.796} C_VEL
LIN {X 0,Y 759.891,Z 638.008,A -85,B 0,C 180,E1 36411.894,E2 36411.894} C_VEL
LIN {X 0,Y 759.895,Z 638.011,A -85,B 0,C 180,E1 36409.161,E2 36409.161} C_VEL
LIN {X 0,Y 759.918,Z 638.008,A -85,B 0,C 180,E1 36406.31,E2 36406.31} C_VEL
LIN {X 0,Y 759.909,Z 638.005,A -85,B 0,C 180,E1 36403.278,E2 36403.278} C_VEL
LIN {X 0,Y 759.911,Z 638.011,A -85,B 0,C 180,E1 36400.344,E2 36400.344} C_VEL
LIN {X 0,Y 759.905,Z 638.015,A -85,B 0,C 180,E1 36398.179,E2 36398.179} C_VEL
LIN {X 0,Y 759.892,Z 680.529,A -85,B 0,C 180,E1 36395.378,E2 36395.378} C_VEL
LIN {X 0,Y 759.911,Z 723.122,A -85,B 0,C 180,E1 36392.693,E2 36392.693} C_VEL
LIN {X 0,Y 759.918,Z 771.919,A -85,B 0,C 180,E1 36389.69,E2 36389.69} C_VEL
LIN {X 0,Y 759.892,Z 818.751,A -85,B 0,C 180,E1 36386.862,E2 36386.862} C_VEL
LIN {X 0,Y 759.894,Z 865.592,A -85,B 0,C 180,E1 36384.074,E2 36384.074} C_VEL
LIN {X 0,Y 759.913,Z 891.644,A -85,B 0,C 180,E1 36382.557,E2 36382.557} C_VEL
LIN {X 0,Y 759.912,Z 1033.648,A -85,B 0,C 180,E1 36381.193,E2 36381.193} C_VEL
LIN {X 0,Y 759.909,Z 1050.134,A -85,B 0,C 180,E1 36380.891,E2 36380.891} C_VEL
LIN {X 0,Y 759.905,Z 1065.295,A -85,B 0,C 180,E1 36380.475,E2 36380.475} C_VEL
LIN {X 0,Y 759.891,Z 1079.991,A -85,B 0,C 180,E1 36379.926,E2 36379.926} C_VEL
LIN {X 0,Y 759.919,Z 1094.151,A -85,B 0,C 180,E1 36379.245,E2 36379.245} C_VEL
LIN {X 0,Y 759.919,Z 1106.654,A -85,B 0,C 180,E1 36378.488,E2 36378.488} C_VEL
LIN {X 0,Y 759.918,Z 1119.23,A -85,B 0,C 180,E1 36377.537,E2 36377.537} C_VEL
LIN {X 0,Y 759.91,Z 1129.191,A -85,B 0,C 180,E1 36376.591,E2 36376.591} C_VEL
LIN {X 0,Y 759.917,Z 1138.401,A -85,B 0,C 180,E1 36375.492,E2 36375.492} C_VEL
LIN {X 0,Y 759.915,Z 1145.49,A -85,B 0,C 180,E1 36374.4,E2 36374.4} C_VEL
LIN {X 0,Y 759.916,Z 1151.258,A -85,B 0,C 180,E1 36373.182,E2 36373.182} C_VEL
LIN {X 0,Y 759.918,Z 1155.035,A -85,B 0,C 180,E1 36371.999,E2 36371.999} C_VEL
LIN {X 0,Y 759.919,Z 1157.083,A -85,B 0,C 180,E1 36370.769,E2 36370.769} C_VEL
LIN {X 0,Y 759.916,Z 1157.385,A -85,B 0,C 180,E1 36369.543,E2 36369.543} C_VEL
LIN {X 0,Y 759.917,Z 1155.909,A -85,B 0,C 180,E1 36368.322,E2 36368.322} C_VEL
LIN {X 0,Y 759.916,Z 1152.648,A -85,B 0,C 180,E1 36367.105,E2 36367.105} C_VEL
LIN {X 0,Y 759.915,Z 1147.569,A -85,B 0,C 180,E1 36365.899,E2 36365.899} C_VEL
LIN {X 0,Y 759.917,Z 1140.778,A -85,B 0,C 180,E1 36364.755,E2 36364.755} C_VEL
LIN {X 0,Y 759.917,Z 1132.633,A -85,B 0,C 180,E1 36363.697,E2 36363.697} C_VEL
LIN {X 0,Y 759.919,Z 1123.064,A -85,B 0,C 180,E1 36362.715,E2 36362.715} C_VEL
LIN {X 0,Y 759.919,Z 1111.108,A -85,B 0,C 180,E1 36361.734,E2 36361.734} C_VEL
LIN {X 0,Y 759.919,Z 1098.393,A -85,B 0,C 180,E1 36360.905,E2 36360.905} C_VEL
LIN {X 0,Y 759.893,Z 1084.651,A -85,B 0,C 180,E1 36360.188,E2 36360.188} C_VEL
LIN {X 0,Y 759.905,Z 1070.801,A -85,B 0,C 180,E1 36359.623,E2 36359.623} C_VEL
LIN {X 0,Y 759.914,Z 1055.493,A -85,B 0,C 180,E1 36359.152,E2 36359.152} C_VEL
LIN {X 0,Y 759.902,Z 1039.867,A -85,B 0,C 180,E1 36358.813,E2 36358.813} C_VEL
LIN {X 0,Y 759.909,Z 1022.948,A -85,B 0,C 180,E1 36358.596,E2 36358.596} C_VEL
LIN {X 0,Y 759.917,Z 891.12,A -85,B 0,C 180,E1 36357.342,E2 36357.342} C_VEL
LIN {X 0,Y 759.906,Z 841.581,A -85,B 0,C 180,E1 36354.412,E2 36354.412} C_VEL
LIN {X 0,Y 759.894,Z 794.706,A -85,B 0,C 180,E1 36351.601,E2 36351.601} C_VEL
LIN {X 0,Y 759.899,Z 749.499,A -85,B 0,C 180,E1 36348.847,E2 36348.847} C_VEL
LIN {X 0,Y 759.915,Z 702.843,A -85,B 0,C 180,E1 36345.95,E2 36345.95} C_VEL
LIN {X 0,Y 759.903,Z 684.179,A -85,B 0,C 180,E1 36344.742,E2 36344.742} C_VEL
LIN {X 0,Y 759.902,Z 645.56,A -85,B 0,C 180,E1 36341.988,E2 36341.988} C_VEL
LIN {X 0,Y 759.892,Z 638.01,A -85,B 0,C 180,E1 36341.432,E2 36341.432} C_VEL
LIN {X 0,Y 759.912,Z 638.014,A -85,B 0,C 180,E1 36338.544,E2 36338.544} C_VEL
LIN {X 0,Y 759.916,Z 638,A -85,B 0,C 180,E1 36335.514,E2 36335.514} C_VEL
LIN {X 0,Y 759.913,Z 638.014,A -85,B 0,C 180,E1 36332.475,E2 36332.475} C_VEL
LIN {X 0,Y 759.899,Z 638.003,A -85,B 0,C 180,E1 36329.523,E2 36329.523} C_VEL
LIN {X 0,Y 759.89,Z 638.007,A -85,B 0,C 180,E1 36326.722,E2 36326.722} C_VEL
LIN {X 0,Y 759.899,Z 638.011,A -85,B 0,C 180,E1 36323.879,E2 36323.879} C_VEL
LIN {X 0,Y 759.912,Z 638.001,A -85,B 0,C 180,E1 36320.922,E2 36320.922} C_VEL
LIN {X 0,Y 759.916,Z 638.015,A -85,B 0,C 180,E1 36317.908,E2 36317.908} C_VEL
LIN {X 0,Y 759.901,Z 638.003,A -85,B 0,C 180,E1 36314.935,E2 36314.935} C_VEL
LIN {X 0,Y 759.896,Z 638.01,A -85,B 0,C 180,E1 36312.087,E2 36312.087} C_VEL
LIN {X 0,Y 759.888,Z 638.157,A -85,B 0,C 180,E1 36311.039,E2 36311.039} C_VEL
LIN {X 0,Y 759.918,Z 689.861,A -85,B 0,C 180,E1 36308.583,E2 36308.583} C_VEL
LIN {X 0,Y 759.914,Z 737.406,A -85,B 0,C 180,E1 36306.364,E2 36306.364} C_VEL
LIN {X 0,Y 759.899,Z 750.967,A -85,B 0,C 180,E1 36305.592,E2 36305.592} C_VEL
LIN {X 0,Y 759.906,Z 760.349,A -85,B 0,C 180,E1 36304.914,E2 36304.914} C_VEL
LIN {X 0,Y 759.918,Z 765.835,A -85,B 0,C 180,E1 36304.364,E2 36304.364} C_VEL
LIN {X 0,Y 759.892,Z 768.112,A -85,B 0,C 180,E1 36304.001,E2 36304.001} C_VEL
LIN {X 0,Y 759.889,Z 768.677,A -85,B 0,C 180,E1 36303.728,E2 36303.728} C_VEL
LIN {X 0,Y 759.903,Z 767.692,A -85,B 0,C 180,E1 36303.464,E2 36303.464} C_VEL
LIN {X 0,Y 759.914,Z 765.278,A -85,B 0,C 180,E1 36303.275,E2 36303.275} C_VEL
LIN {X 0,Y 759.916,Z 760.408,A -85,B 0,C 180,E1 36303.117,E2 36303.117} C_VEL
LIN {X 0,Y 759.912,Z 752.908,A -85,B 0,C 180,E1 36303.045,E2 36303.045} C_VEL
LIN {X 0,Y 759.911,Z 638.015,A -85,B 0,C 180,E1 36303.029,E2 36303.029} C_VEL
LIN {X 0,Y 759.898,Z 638.037,A -85,B 0,C 180,E1 36300.983,E2 36300.983} C_VEL
LIN {X 0,Y 759.898,Z 693.683,A -85,B 0,C 180,E1 36298.323,E2 36298.323} C_VEL
LIN {X 0,Y 759.891,Z 750.994,A -85,B 0,C 180,E1 36295.651,E2 36295.651} C_VEL
LIN {X 0,Y 759.89,Z 757.368,A -85,B 0,C 180,E1 36295.358,E2 36295.358} C_VEL
LIN {X 0,Y 759.911,Z 1023.044,A -85,B 0,C 180,E1 36292.665,E2 36292.665} C_VEL
LIN {X 0,Y 759.906,Z 1065.118,A -85,B 0,C 180,E1 36292.216,E2 36292.216} C_VEL
LIN {X 0,Y 759.915,Z 1085.837,A -85,B 0,C 180,E1 36291.86,E2 36291.86} C_VEL
LIN {X 0,Y 759.905,Z 1107.869,A -85,B 0,C 180,E1 36291.344,E2 36291.344} C_VEL
LIN {X 0,Y 759.911,Z 1128.402,A -85,B 0,C 180,E1 36290.728,E2 36290.728} C_VEL
LIN {X 0,Y 759.919,Z 1147.754,A -85,B 0,C 180,E1 36290.004,E2 36290.004} C_VEL
LIN {X 0,Y 759.918,Z 1167.542,A -85,B 0,C 180,E1 36289.124,E2 36289.124} C_VEL
LIN {X 0,Y 759.913,Z 1186.47,A -85,B 0,C 180,E1 36288.129,E2 36288.129} C_VEL
LIN {X 0,Y 759.916,Z 1204.303,A -85,B 0,C 180,E1 36287.022,E2 36287.022} C_VEL
LIN {X 0,Y 759.918,Z 1221.192,A -85,B 0,C 180,E1 36285.804,E2 36285.804} C_VEL
LIN {X 0,Y 759.911,Z 1237.484,A -85,B 0,C 180,E1 36284.434,E2 36284.434} C_VEL
LIN {X 0,Y 759.906,Z 1251.341,A -85,B 0,C 180,E1 36283.079,E2 36283.079} C_VEL
LIN {X 0,Y 759.911,Z 1263.467,A -85,B 0,C 180,E1 36281.69,E2 36281.69} C_VEL
LIN {X 0,Y 759.903,Z 1274.587,A -85,B 0,C 180,E1 36280.188,E2 36280.188} C_VEL
LIN {X 0,Y 759.909,Z 1283.855,A -85,B 0,C 180,E1 36278.702,E2 36278.702} C_VEL
LIN {X 0,Y 759.918,Z 1291.53,A -85,B 0,C 180,E1 36277.18,E2 36277.18} C_VEL
LIN {X 0,Y 759.907,Z 1298.148,A -85,B 0,C 180,E1 36275.511,E2 36275.511} C_VEL
LIN {X 0,Y 759.901,Z 1302.827,A -85,B 0,C 180,E1 36273.922,E2 36273.922} C_VEL
LIN {X 0,Y 759.899,Z 1305.785,A -85,B 0,C 180,E1 36272.337,E2 36272.337} C_VEL
LIN {X 0,Y 759.9,Z 1307.33,A -85,B 0,C 180,E1 36270.602,E2 36270.602} C_VEL
LIN {X 0,Y 759.919,Z 1307.209,A -85,B 0,C 180,E1 36269.019,E2 36269.019} C_VEL
LIN {X 0,Y 759.917,Z 1305.335,A -85,B 0,C 180,E1 36267.359,E2 36267.359} C_VEL
LIN {X 0,Y 759.907,Z 1301.805,A -85,B 0,C 180,E1 36265.698,E2 36265.698} C_VEL
LIN {X 0,Y 759.898,Z 1296.869,A -85,B 0,C 180,E1 36264.108,E2 36264.108} C_VEL
LIN {X 0,Y 759.908,Z 1290.107,A -85,B 0,C 180,E1 36262.514,E2 36262.514} C_VEL
LIN {X 0,Y 759.912,Z 1281.588,A -85,B 0,C 180,E1 36260.914,E2 36260.914} C_VEL
LIN {X 0,Y 759.909,Z 1271.682,A -85,B 0,C 180,E1 36259.384,E2 36259.384} C_VEL
LIN {X 0,Y 759.912,Z 1260.252,A -85,B 0,C 180,E1 36257.923,E2 36257.923} C_VEL
LIN {X 0,Y 759.917,Z 1246.77,A -85,B 0,C 180,E1 36256.454,E2 36256.454} C_VEL
LIN {X 0,Y 759.911,Z 1232.64,A -85,B 0,C 180,E1 36255.132,E2 36255.132} C_VEL
LIN {X 0,Y 759.911,Z 1216.728,A -85,B 0,C 180,E1 36253.85,E2 36253.85} C_VEL
LIN {X 0,Y 759.913,Z 1199.444,A -85,B 0,C 180,E1 36252.66,E2 36252.66} C_VEL
LIN {X 0,Y 759.916,Z 1181.354,A -85,B 0,C 180,E1 36251.591,E2 36251.591} C_VEL
LIN {X 0,Y 759.916,Z 1162.49,A -85,B 0,C 180,E1 36250.635,E2 36250.635} C_VEL
LIN {X 0,Y 759.919,Z 1142.727,A -85,B 0,C 180,E1 36249.793,E2 36249.793} C_VEL
LIN {X 0,Y 759.91,Z 1123.088,A -85,B 0,C 180,E1 36249.103,E2 36249.103} C_VEL
LIN {X 0,Y 759.904,Z 1102.447,A -85,B 0,C 180,E1 36248.511,E2 36248.511} C_VEL
LIN {X 0,Y 759.913,Z 1081.567,A -85,B 0,C 180,E1 36248.056,E2 36248.056} C_VEL
LIN {X 0,Y 759.907,Z 1059.604,A -85,B 0,C 180,E1 36247.716,E2 36247.716} C_VEL
LIN {X 0,Y 759.901,Z 777.506,A -85,B 0,C 180,E1 36244.848,E2 36244.848} C_VEL
LIN {X 0,Y 759.89,Z 757.295,A -85,B 0,C 180,E1 36244.639,E2 36244.639} C_VEL
LIN {X 0,Y 759.91,Z 698.322,A -85,B 0,C 180,E1 36241.896,E2 36241.896} C_VEL
LIN {X 0,Y 759.89,Z 642.071,A -85,B 0,C 180,E1 36239.212,E2 36239.212} C_VEL
LIN {X 0,Y 759.9,Z 638.013,A -85,B 0,C 180,E1 36238.992,E2 36238.992} C_VEL
LIN {X 0,Y 759.912,Z 638.016,A -85,B 0,C 180,E1 36236.957,E2 36236.957} C_VEL
LIN {X 0,Y 759.912,Z 755.764,A -85,B 0,C 180,E1 36236.942,E2 36236.942} C_VEL
LIN {X 0,Y 759.913,Z 762.449,A -85,B 0,C 180,E1 36236.835,E2 36236.835} C_VEL
LIN {X 0,Y 759.914,Z 766.172,A -85,B 0,C 180,E1 36236.671,E2 36236.671} C_VEL
LIN {X 0,Y 759.897,Z 768.234,A -85,B 0,C 180,E1 36236.451,E2 36236.451} C_VEL
LIN {X 0,Y 759.888,Z 768.626,A -85,B 0,C 180,E1 36236.178,E2 36236.178} C_VEL
LIN {X 0,Y 759.904,Z 767.134,A -85,B 0,C 180,E1 36235.815,E2 36235.815} C_VEL
LIN {X 0,Y 759.915,Z 762.389,A -85,B 0,C 180,E1 36235.268,E2 36235.268} C_VEL
LIN {X 0,Y 759.914,Z 754.191,A -85,B 0,C 180,E1 36234.623,E2 36234.623} C_VEL
LIN {X 0,Y 759.894,Z 741.99,A -85,B 0,C 180,E1 36233.879,E2 36233.879} C_VEL
LIN {X 0,Y 759.913,Z 687.887,A -85,B 0,C 180,E1 36231.165,E2 36231.165} C_VEL
LIN {X 0,Y 759.907,Z 638.833,A -85,B 0,C 180,E1 36228.625,E2 36228.625} C_VEL
LIN {X 0,Y 759.903,Z 638.015,A -85,B 0,C 180,E1 36228.558,E2 36228.558} C_VEL
LIN {X 0,Y 759.9,Z 638.012,A -85,B 0,C 180,E1 36225.677,E2 36225.677} C_VEL
LIN {X 0,Y 759.894,Z 638.012,A -85,B 0,C 180,E1 36222.868,E2 36222.868} C_VEL
LIN {X 0,Y 759.908,Z 638.011,A -85,B 0,C 180,E1 36219.95,E2 36219.95} C_VEL
LIN {X 0,Y 759.913,Z 638.013,A -85,B 0,C 180,E1 36216.995,E2 36216.995} C_VEL
LIN {X 0,Y 759.909,Z 638.015,A -85,B 0,C 180,E1 36214.093,E2 36214.093} C_VEL
LIN {X 0,Y 759.902,Z 638.013,A -85,B 0,C 180,E1 36211.227,E2 36211.227} C_VEL
LIN {X 0,Y 759.898,Z 638.183,A -85,B 0,C 180,E1 36209.894,E2 36209.894} C_VEL
LIN {X 0,Y 759.899,Z 674.226,A -85,B 0,C 180,E1 36207.19,E2 36207.19} C_VEL
LIN {X 0,Y 759.9,Z 700.569,A -85,B 0,C 180,E1 36205.28,E2 36205.28} C_VEL
LIN {X 0,Y 759.917,Z 985.87,A -85,B 0,C 180,E1 36202.391,E2 36202.391} C_VEL
LIN {X 0,Y 759.909,Z 1009.319,A -85,B 0,C 180,E1 36202.106,E2 36202.106} C_VEL
LIN {X 0,Y 759.913,Z 1030.271,A -85,B 0,C 180,E1 36201.728,E2 36201.728} C_VEL
LIN {X 0,Y 759.91,Z 1050.97,A -85,B 0,C 180,E1 36201.214,E2 36201.214} C_VEL
LIN {X 0,Y 759.906,Z 1071.637,A -85,B 0,C 180,E1 36200.568,E2 36200.568} C_VEL
LIN {X 0,Y 759.918,Z 1091.927,A -85,B 0,C 180,E1 36199.79,E2 36199.79} C_VEL
LIN {X 0,Y 759.916,Z 1111.023,A -85,B 0,C 180,E1 36198.905,E2 36198.905} C_VEL
LIN {X 0,Y 759.916,Z 1130.339,A -85,B 0,C 180,E1 36197.853,E2 36197.853} C_VEL
LIN {X 0,Y 759.912,Z 1147.734,A -85,B 0,C 180,E1 36196.748,E2 36196.748} C_VEL
LIN {X 0,Y 759.911,Z 1164.638,A -85,B 0,C 180,E1 36195.492,E2 36195.492} C_VEL
LIN {X 0,Y 759.91,Z 1179.066,A -85,B 0,C 180,E1 36194.244,E2 36194.244} C_VEL
LIN {X 0,Y 759.912,Z 1193.138,A -85,B 0,C 180,E1 36192.837,E2 36192.837} C_VEL
LIN {X 0,Y 759.908,Z 1205.585,A -85,B 0,C 180,E1 36191.383,E2 36191.383} C_VEL
LIN {X 0,Y 759.917,Z 1216.053,A -85,B 0,C 180,E1 36189.926,E2 36189.926} C_VEL
LIN {X 0,Y 759.899,Z 1225.638,A -85,B 0,C 180,E1 36188.322,E2 36188.322} C_VEL
LIN {X 0,Y 759.917,Z 1233.068,A -85,B 0,C 180,E1 36186.801,E2 36186.801} C_VEL
LIN {X 0,Y 759.91,Z 1239.007,A -85,B 0,C 180,E1 36185.209,E2 36185.209} C_VEL
LIN {X 0,Y 759.914,Z 1243.685,A -85,B 0,C 180,E1 36183.47,E2 36183.47} C_VEL
LIN {X 0,Y 759.912,Z 1246.442,A -85,B 0,C 180,E1 36181.81,E2 36181.81} C_VEL
LIN {X 0,Y 759.906,Z 1247.449,A -85,B 0,C 180,E1 36180.151,E2 36180.151} C_VEL
LIN {X 0,Y 759.911,Z 1246.787,A -85,B 0,C 180,E1 36178.492,E2 36178.492} C_VEL
LIN {X 0,Y 759.904,Z 1244.988,A -85,B 0,C 180,E1 36177.08,E2 36177.08} C_VEL
LIN {X 0,Y 758.895,Z 1243.979,A -85,B 0,C 180,E1 36176.505,E2 36176.505} C_VEL
LIN {X 0,Y 752.564,Z 1240.001,A -85,B 0,C 180,E1 36174.949,E2 36174.949} C_VEL
LIN {X 0,Y 751.915,Z 1238.521,A -85,B 0,C 180,E1 36174.498,E2 36174.498} C_VEL
LIN {X 0,Y 751.924,Z 1232.438,A -85,B 0,C 180,E1 36172.896,E2 36172.896} C_VEL
LIN {X 0,Y 751.918,Z 1224.897,A -85,B 0,C 180,E1 36171.358,E2 36171.358} C_VEL
LIN {X 0,Y 751.93,Z 1215.172,A -85,B 0,C 180,E1 36169.745,E2 36169.745} C_VEL
LIN {X 0,Y 751.951,Z 1204.466,A -85,B 0,C 180,E1 36168.261,E2 36168.261} C_VEL
LIN {X 0,Y 751.982,Z 1192.441,A -85,B 0,C 180,E1 36166.857,E2 36166.857} C_VEL
LIN {X 0,Y 752.014,Z 1178.347,A -85,B 0,C 180,E1 36165.446,E2 36165.446} C_VEL
LIN {X 0,Y 752.064,Z 1162.761,A -85,B 0,C 180,E1 36164.104,E2 36164.104} C_VEL
LIN {X 0,Y 752.123,Z 1146.161,A -85,B 0,C 180,E1 36162.874,E2 36162.874} C_VEL
LIN {X 0,Y 752.167,Z 1128.525,A -85,B 0,C 180,E1 36161.756,E2 36161.756} C_VEL
LIN {X 0,Y 752.231,Z 1110.005,A -85,B 0,C 180,E1 36160.752,E2 36160.752} C_VEL
LIN {X 0,Y 752.302,Z 1090.805,A -85,B 0,C 180,E1 36159.865,E2 36159.865} C_VEL
LIN {X 0,Y 752.336,Z 1070.882,A -85,B 0,C 180,E1 36159.097,E2 36159.097} C_VEL
LIN {X 0,Y 752.409,Z 1050.208,A -85,B 0,C 180,E1 36158.453,E2 36158.453} C_VEL
LIN {X 0,Y 752.46,Z 1028.677,A -85,B 0,C 180,E1 36157.923,E2 36157.923} C_VEL
LIN {X 0,Y 752.486,Z 1007.419,A -85,B 0,C 180,E1 36157.543,E2 36157.543} C_VEL
LIN {X 0,Y 752.52,Z 977.267,A -85,B 0,C 180,E1 36157.199,E2 36157.199} C_VEL
LIN {X 0,Y 752.648,Z 701.616,A -85,B 0,C 180,E1 36154.379,E2 36154.379} C_VEL
LIN {X 0,Y 752.347,Z 699.786,A -85,B 0,C 180,E1 36154.325,E2 36154.325} C_VEL
LIN {X 0,Y 752.437,Z 660.279,A -85,B 0,C 180,E1 36151.376,E2 36151.376} C_VEL
LIN {X 0,Y 752.422,Z 640.883,A -85,B 0,C 180,E1 36149.896,E2 36149.896} C_VEL
LIN {X 0,Y 751.952,Z 639.004,A -85,B 0,C 180,E1 36149.715,E2 36149.715} C_VEL
LIN {X 0,Y 751.954,Z 638.998,A -85,B 0,C 180,E1 36146.901,E2 36146.901} C_VEL
LIN {X 0,Y 751.98,Z 639.002,A -85,B 0,C 180,E1 36144.005,E2 36144.005} C_VEL
LIN {X 0,Y 751.977,Z 638.994,A -85,B 0,C 180,E1 36141.028,E2 36141.028} C_VEL
LIN {X 0,Y 751.972,Z 638.995,A -85,B 0,C 180,E1 36138.014,E2 36138.014} C_VEL
LIN {X 0,Y 751.975,Z 639.003,A -85,B 0,C 180,E1 36135.084,E2 36135.084} C_VEL
LIN {X 0,Y 751.953,Z 638.996,A -85,B 0,C 180,E1 36132.287,E2 36132.287} C_VEL
LIN {X 0,Y 751.968,Z 639,A -85,B 0,C 180,E1 36129.416,E2 36129.416} C_VEL
LIN {X 0,Y 751.965,Z 638.997,A -85,B 0,C 180,E1 36126.564,E2 36126.564} C_VEL
LIN {X 0,Y 751.954,Z 638.997,A -85,B 0,C 180,E1 36123.676,E2 36123.676} C_VEL
LIN {X 0,Y 751.975,Z 639.004,A -85,B 0,C 180,E1 36120.793,E2 36120.793} C_VEL
LIN {X 0,Y 751.963,Z 638.995,A -85,B 0,C 180,E1 36117.909,E2 36117.909} C_VEL
LIN {X 0,Y 751.976,Z 638.995,A -85,B 0,C 180,E1 36114.926,E2 36114.926} C_VEL
LIN {X 0,Y 751.964,Z 639.002,A -85,B 0,C 180,E1 36112.024,E2 36112.024} C_VEL
LIN {X 0,Y 751.951,Z 638.996,A -85,B 0,C 180,E1 36109.175,E2 36109.175} C_VEL
LIN {X 0,Y 751.959,Z 639.003,A -85,B 0,C 180,E1 36106.374,E2 36106.374} C_VEL
LIN {X 0,Y 751.973,Z 638.995,A -85,B 0,C 180,E1 36103.457,E2 36103.457} C_VEL
LIN {X 0,Y 751.975,Z 638.994,A -85,B 0,C 180,E1 36100.419,E2 36100.419} C_VEL
LIN {X 0,Y 751.968,Z 639.001,A -85,B 0,C 180,E1 36097.412,E2 36097.412} C_VEL
LIN {X 0,Y 751.951,Z 638.998,A -85,B 0,C 180,E1 36094.577,E2 36094.577} C_VEL
LIN {X 0,Y 751.958,Z 638.998,A -85,B 0,C 180,E1 36091.83,E2 36091.83} C_VEL
LIN {X 0,Y 751.974,Z 638.998,A -85,B 0,C 180,E1 36089.011,E2 36089.011} C_VEL
LIN {X 0,Y 751.962,Z 638.994,A -85,B 0,C 180,E1 36086.036,E2 36086.036} C_VEL
LIN {X 0,Y 751.955,Z 639.003,A -85,B 0,C 180,E1 36083.205,E2 36083.205} C_VEL
LIN {X 0,Y 751.962,Z 638.996,A -85,B 0,C 180,E1 36080.433,E2 36080.433} C_VEL
LIN {X 0,Y 751.975,Z 638.995,A -85,B 0,C 180,E1 36077.484,E2 36077.484} C_VEL
LIN {X 0,Y 751.968,Z 639.002,A -85,B 0,C 180,E1 36074.579,E2 36074.579} C_VEL
LIN {X 0,Y 751.951,Z 638.996,A -85,B 0,C 180,E1 36071.701,E2 36071.701} C_VEL
LIN {X 0,Y 751.963,Z 639.003,A -85,B 0,C 180,E1 36068.961,E2 36068.961} C_VEL
LIN {X 0,Y 751.976,Z 638.995,A -85,B 0,C 180,E1 36066.076,E2 36066.076} C_VEL
LIN {X 0,Y 751.978,Z 638.993,A -85,B 0,C 180,E1 36062.985,E2 36062.985} C_VEL
LIN {X 0,Y 751.967,Z 639.001,A -85,B 0,C 180,E1 36059.956,E2 36059.956} C_VEL
LIN {X 0,Y 751.952,Z 638.997,A -85,B 0,C 180,E1 36057.146,E2 36057.146} C_VEL
LIN {X 0,Y 751.956,Z 638.997,A -85,B 0,C 180,E1 36054.337,E2 36054.337} C_VEL
LIN {X 0,Y 751.979,Z 638.999,A -85,B 0,C 180,E1 36051.519,E2 36051.519} C_VEL
LIN {X 0,Y 751.972,Z 638.994,A -85,B 0,C 180,E1 36048.471,E2 36048.471} C_VEL
LIN {X 0,Y 751.959,Z 638.999,A -85,B 0,C 180,E1 36045.515,E2 36045.515} C_VEL
LIN {X 0,Y 751.952,Z 639,A -85,B 0,C 180,E1 36042.779,E2 36042.779} C_VEL
LIN {X 0,Y 751.965,Z 638.997,A -85,B 0,C 180,E1 36039.896,E2 36039.896} C_VEL
LIN {X 0,Y 751.981,Z 639.138,A -85,B 0,C 180,E1 36038.469,E2 36038.469} C_VEL
LIN {X 0,Y 752.627,Z 642.651,A -85,B 0,C 180,E1 36038.202,E2 36038.202} C_VEL
LIN {X 0,Y 752.523,Z 687.026,A -85,B 0,C 180,E1 36035.263,E2 36035.263} C_VEL
LIN {X 0,Y 752.302,Z 724.668,A -85,B 0,C 180,E1 36032.839,E2 36032.839} C_VEL
LIN {X 0,Y 752.214,Z 773.373,A -85,B 0,C 180,E1 36029.811,E2 36029.811} C_VEL
LIN {X 0,Y 752.111,Z 820.129,A -85,B 0,C 180,E1 36026.958,E2 36026.958} C_VEL
LIN {X 0,Y 752.048,Z 866.432,A -85,B 0,C 180,E1 36024.174,E2 36024.174} C_VEL
LIN {X 0,Y 752.073,Z 891.662,A -85,B 0,C 180,E1 36022.69,E2 36022.69} C_VEL
LIN {X 0,Y 752.062,Z 1033.775,A -85,B 0,C 180,E1 36021.31,E2 36021.31} C_VEL
LIN {X 0,Y 752.045,Z 1051.014,A -85,B 0,C 180,E1 36020.987,E2 36020.987} C_VEL
LIN {X 0,Y 752.018,Z 1066.368,A -85,B 0,C 180,E1 36020.55,E2 36020.55} C_VEL
LIN {X 0,Y 751.982,Z 1081.12,A -85,B 0,C 180,E1 36019.982,E2 36019.982} C_VEL
LIN {X 0,Y 751.99,Z 1094.298,A -85,B 0,C 180,E1 36019.335,E2 36019.335} C_VEL
LIN {X 0,Y 751.968,Z 1107.361,A -85,B 0,C 180,E1 36018.53,E2 36018.53} C_VEL
LIN {X 0,Y 751.948,Z 1119.841,A -85,B 0,C 180,E1 36017.563,E2 36017.563} C_VEL
LIN {X 0,Y 751.927,Z 1129.625,A -85,B 0,C 180,E1 36016.613,E2 36016.613} C_VEL
LIN {X 0,Y 751.926,Z 1138.163,A -85,B 0,C 180,E1 36015.582,E2 36015.582} C_VEL
LIN {X 0,Y 751.921,Z 1145.328,A -85,B 0,C 180,E1 36014.478,E2 36014.478} C_VEL
LIN {X 0,Y 751.919,Z 1151.238,A -85,B 0,C 180,E1 36013.222,E2 36013.222} C_VEL
LIN {X 0,Y 751.918,Z 1154.954,A -85,B 0,C 180,E1 36012.051,E2 36012.051} C_VEL
LIN {X 0,Y 751.918,Z 1157.057,A -85,B 0,C 180,E1 36010.807,E2 36010.807} C_VEL
LIN {X 0,Y 751.916,Z 1157.372,A -85,B 0,C 180,E1 36009.491,E2 36009.491} C_VEL
LIN {X 0,Y 751.918,Z 1155.812,A -85,B 0,C 180,E1 36008.257,E2 36008.257} C_VEL
LIN {X 0,Y 751.917,Z 1152.49,A -85,B 0,C 180,E1 36007.027,E2 36007.027} C_VEL
LIN {X 0,Y 751.917,Z 1147.667,A -85,B 0,C 180,E1 36005.877,E2 36005.877} C_VEL
LIN {X 0,Y 751.924,Z 1140.982,A -85,B 0,C 180,E1 36004.729,E2 36004.729} C_VEL
LIN {X 0,Y 751.933,Z 1132.242,A -85,B 0,C 180,E1 36003.583,E2 36003.583} C_VEL
LIN {X 0,Y 751.945,Z 1122.538,A -85,B 0,C 180,E1 36002.591,E2 36002.591} C_VEL
LIN {X 0,Y 751.964,Z 1110.483,A -85,B 0,C 180,E1 36001.6,E2 36001.6} C_VEL
LIN {X 0,Y 751.985,Z 1096.95,A -85,B 0,C 180,E1 36000.724,E2 36000.724} C_VEL
LIN {X 0,Y 751.978,Z 1083.637,A -85,B 0,C 180,E1 36000.038,E2 36000.038} C_VEL
LIN {X 0,Y 752.021,Z 1069.445,A -85,B 0,C 180,E1 35999.467,E2 35999.467} C_VEL
LIN {X 0,Y 752.039,Z 1053.71,A -85,B 0,C 180,E1 35998.991,E2 35998.991} C_VEL
LIN {X 0,Y 752.051,Z 1037.328,A -85,B 0,C 180,E1 35998.652,E2 35998.652} C_VEL
LIN {X 0,Y 752.072,Z 1014.649,A -85,B 0,C 180,E1 35998.397,E2 35998.397} C_VEL
LIN {X 0,Y 752.035,Z 890.988,A -85,B 0,C 180,E1 35997.199,E2 35997.199} C_VEL
LIN {X 0,Y 752.095,Z 842.093,A -85,B 0,C 180,E1 35994.277,E2 35994.277} C_VEL
LIN {X 0,Y 752.151,Z 794.594,A -85,B 0,C 180,E1 35991.399,E2 35991.399} C_VEL
LIN {X 0,Y 752.235,Z 750.026,A -85,B 0,C 180,E1 35988.654,E2 35988.654} C_VEL
LIN {X 0,Y 752.418,Z 708.705,A -85,B 0,C 180,E1 35986.043,E2 35986.043} C_VEL
LIN {X 0,Y 752.921,Z 682.813,A -85,B 0,C 180,E1 35984.242,E2 35984.242} C_VEL
LIN {X 0,Y 753.057,Z 644.752,A -85,B 0,C 180,E1 35981.498,E2 35981.498} C_VEL
LIN {X 0,Y 752.809,Z 641.738,A -85,B 0,C 180,E1 35981.259,E2 35981.259} C_VEL
LIN {X 0,Y 751.96,Z 639.005,A -85,B 0,C 180,E1 35980.978,E2 35980.978} C_VEL
LIN {X 0,Y 751.953,Z 638.998,A -85,B 0,C 180,E1 35978.141,E2 35978.141} C_VEL
LIN {X 0,Y 751.96,Z 638.993,A -85,B 0,C 180,E1 35975.321,E2 35975.321} C_VEL
LIN {X 0,Y 751.973,Z 639.004,A -85,B 0,C 180,E1 35972.35,E2 35972.35} C_VEL
LIN {X 0,Y 751.972,Z 638.991,A -85,B 0,C 180,E1 35969.348,E2 35969.348} C_VEL
LIN {X 0,Y 751.969,Z 639.003,A -85,B 0,C 180,E1 35966.325,E2 35966.325} C_VEL
LIN {X 0,Y 751.953,Z 638.995,A -85,B 0,C 180,E1 35963.429,E2 35963.429} C_VEL
LIN {X 0,Y 751.955,Z 638.995,A -85,B 0,C 180,E1 35960.633,E2 35960.633} C_VEL
LIN {X 0,Y 751.969,Z 639.002,A -85,B 0,C 180,E1 35957.783,E2 35957.783} C_VEL
LIN {X 0,Y 751.974,Z 638.991,A -85,B 0,C 180,E1 35954.76,E2 35954.76} C_VEL
LIN {X 0,Y 751.974,Z 639.004,A -85,B 0,C 180,E1 35951.758,E2 35951.758} C_VEL
LIN {X 0,Y 751.98,Z 639.16,A -85,B 0,C 180,E1 35951.372,E2 35951.372} C_VEL
LIN {X 0,Y 752.82,Z 642.331,A -85,B 0,C 180,E1 35951.173,E2 35951.173} C_VEL
LIN {X 0,Y 752.659,Z 694.127,A -85,B 0,C 180,E1 35948.684,E2 35948.684} C_VEL
LIN {X 0,Y 753.033,Z 748.854,A -85,B 0,C 180,E1 35946.123,E2 35946.123} C_VEL
LIN {X 0,Y 754.044,Z 760.945,A -85,B 0,C 180,E1 35945.463,E2 35945.463} C_VEL
LIN {X 0,Y 755.126,Z 768.892,A -85,B 0,C 180,E1 35944.89,E2 35944.89} C_VEL
LIN {X 0,Y 756.18,Z 773.778,A -85,B 0,C 180,E1 35944.374,E2 35944.374} C_VEL
LIN {X 0,Y 757.002,Z 775.915,A -85,B 0,C 180,E1 35943.952,E2 35943.952} C_VEL
LIN {X 0,Y 757.578,Z 776.163,A -85,B 0,C 180,E1 35943.572,E2 35943.572} C_VEL
LIN {X 0,Y 757.78,Z 774.699,A -85,B 0,C 180,E1 35943.221,E2 35943.221} C_VEL
LIN {X 0,Y 757.509,Z 771.586,A -85,B 0,C 180,E1 35942.922,E2 35942.922} C_VEL
LIN {X 0,Y 756.833,Z 766.938,A -85,B 0,C 180,E1 35942.706,E2 35942.706} C_VEL
LIN {X 0,Y 755.904,Z 759.904,A -85,B 0,C 180,E1 35942.574,E2 35942.574} C_VEL
LIN {X 0,Y 755.582,Z 752.135,A -85,B 0,C 180,E1 35942.535,E2 35942.535} C_VEL
LIN {X 0,Y 755.483,Z 644.677,A -85,B 0,C 180,E1 35942.524,E2 35942.524} C_VEL
LIN {X 0,Y 753.074,Z 642.154,A -85,B 0,C 180,E1 35942.235,E2 35942.235} C_VEL
LIN {X 0,Y 752.009,Z 639.28,A -85,B 0,C 180,E1 35942.106,E2 35942.106} C_VEL
LIN {X 0,Y 751.967,Z 638.998,A -85,B 0,C 180,E1 35942.086,E2 35942.086} C_VEL
LIN {X 0,Y 752.009,Z 639.239,A -85,B 0,C 180,E1 35941.286,E2 35941.286} C_VEL
LIN {X 0,Y 752.753,Z 642.12,A -85,B 0,C 180,E1 35941.11,E2 35941.11} C_VEL
LIN {X 0,Y 752.631,Z 697.919,A -85,B 0,C 180,E1 35938.419,E2 35938.419} C_VEL
LIN {X 0,Y 752.482,Z 756.437,A -85,B 0,C 180,E1 35935.668,E2 35935.668} C_VEL
LIN {X 0,Y 752.656,Z 758.995,A -85,B 0,C 180,E1 35935.603,E2 35935.603} C_VEL
LIN {X 0,Y 752.525,Z 1025.589,A -85,B 0,C 180,E1 35932.874,E2 35932.874} C_VEL
LIN {X 0,Y 752.486,Z 1065.631,A -85,B 0,C 180,E1 35932.44,E2 35932.44} C_VEL
LIN {X 0,Y 752.465,Z 1087.545,A -85,B 0,C 180,E1 35932.055,E2 35932.055} C_VEL
LIN {X 0,Y 752.401,Z 1108.423,A -85,B 0,C 180,E1 35931.553,E2 35931.553} C_VEL
LIN {X 0,Y 752.351,Z 1129.696,A -85,B 0,C 180,E1 35930.901,E2 35930.901} C_VEL
LIN {X 0,Y 752.304,Z 1149.752,A -85,B 0,C 180,E1 35930.134,E2 35930.134} C_VEL
LIN {X 0,Y 752.236,Z 1169.154,A -85,B 0,C 180,E1 35929.246,E2 35929.246} C_VEL
LIN {X 0,Y 752.169,Z 1187.823,A -85,B 0,C 180,E1 35928.242,E2 35928.242} C_VEL
LIN {X 0,Y 752.122,Z 1206.115,A -85,B 0,C 180,E1 35927.084,E2 35927.084} C_VEL
LIN {X 0,Y 752.069,Z 1222.71,A -85,B 0,C 180,E1 35925.854,E2 35925.854} C_VEL
LIN {X 0,Y 752.019,Z 1237.987,A -85,B 0,C 180,E1 35924.543,E2 35924.543} C_VEL
LIN {X 0,Y 751.975,Z 1252.051,A -85,B 0,C 180,E1 35923.141,E2 35923.141} C_VEL
LIN {X 0,Y 751.96,Z 1264.748,A -85,B 0,C 180,E1 35921.659,E2 35921.659} C_VEL
LIN {X 0,Y 751.929,Z 1275.333,A -85,B 0,C 180,E1 35920.186,E2 35920.186} C_VEL
LIN {X 0,Y 751.916,Z 1285.078,A -85,B 0,C 180,E1 35918.564,E2 35918.564} C_VEL
LIN {X 0,Y 751.911,Z 1292.938,A -85,B 0,C 180,E1 35916.949,E2 35916.949} C_VEL
LIN {X 0,Y 751.918,Z 1298.906,A -85,B 0,C 180,E1 35915.34,E2 35915.34} C_VEL
LIN {X 0,Y 751.915,Z 1303.628,A -85,B 0,C 180,E1 35913.582,E2 35913.582} C_VEL
LIN {X 0,Y 751.912,Z 1306.417,A -85,B 0,C 180,E1 35911.904,E2 35911.904} C_VEL
LIN {X 0,Y 751.899,Z 1307.418,A -85,B 0,C 180,E1 35910.304,E2 35910.304} C_VEL
LIN {X 0,Y 751.905,Z 1306.883,A -85,B 0,C 180,E1 35908.627,E2 35908.627} C_VEL
LIN {X 0,Y 751.916,Z 1304.727,A -85,B 0,C 180,E1 35906.95,E2 35906.95} C_VEL
LIN {X 0,Y 751.905,Z 1300.782,A -85,B 0,C 180,E1 35905.27,E2 35905.27} C_VEL
LIN {X 0,Y 751.911,Z 1295.063,A -85,B 0,C 180,E1 35903.586,E2 35903.586} C_VEL
LIN {X 0,Y 751.925,Z 1287.909,A -85,B 0,C 180,E1 35901.973,E2 35901.973} C_VEL
LIN {X 0,Y 751.938,Z 1278.827,A -85,B 0,C 180,E1 35900.354,E2 35900.354} C_VEL
LIN {X 0,Y 751.944,Z 1268.798,A -85,B 0,C 180,E1 35898.882,E2 35898.882} C_VEL
LIN {X 0,Y 751.98,Z 1256.97,A -85,B 0,C 180,E1 35897.404,E2 35897.404} C_VEL
LIN {X 0,Y 752.01,Z 1242.899,A -85,B 0,C 180,E1 35895.917,E2 35895.917} C_VEL
LIN {X 0,Y 752.049,Z 1227.848,A -85,B 0,C 180,E1 35894.565,E2 35894.565} C_VEL
LIN {X 0,Y 752.097,Z 1211.124,A -85,B 0,C 180,E1 35893.271,E2 35893.271} C_VEL
LIN {X 0,Y 752.162,Z 1193.075,A -85,B 0,C 180,E1 35892.076,E2 35892.076} C_VEL
LIN {X 0,Y 752.227,Z 1174.719,A -85,B 0,C 180,E1 35891.034,E2 35891.034} C_VEL
LIN {X 0,Y 752.278,Z 1155.376,A -85,B 0,C 180,E1 35890.106,E2 35890.106} C_VEL
LIN {X 0,Y 752.333,Z 1135.123,A -85,B 0,C 180,E1 35889.296,E2 35889.296} C_VEL
LIN {X 0,Y 752.4,Z 1114.81,A -85,B 0,C 180,E1 35888.625,E2 35888.625} C_VEL
LIN {X 0,Y 752.441,Z 1093.672,A -85,B 0,C 180,E1 35888.078,E2 35888.078} C_VEL
LIN {X 0,Y 752.482,Z 1071.742,A -85,B 0,C 180,E1 35887.656,E2 35887.656} C_VEL
LIN {X 0,Y 752.512,Z 1049.289,A -85,B 0,C 180,E1 35887.366,E2 35887.366} C_VEL
LIN {X 0,Y 752.655,Z 777.883,A -85,B 0,C 180,E1 35884.593,E2 35884.593} C_VEL
LIN {X 0,Y 752.48,Z 757.295,A -85,B 0,C 180,E1 35884.372,E2 35884.372} C_VEL
LIN {X 0,Y 752.631,Z 698.322,A -85,B 0,C 180,E1 35881.6,E2 35881.6} C_VEL
LIN {X 0,Y 752.749,Z 642.979,A -85,B 0,C 180,E1 35878.932,E2 35878.932} C_VEL
LIN {X 0,Y 752.554,Z 641.15,A -85,B 0,C 180,E1 35878.833,E2 35878.833} C_VEL
LIN {X 0,Y 751.977,Z 639.004,A -85,B 0,C 180,E1 35878.689,E2 35878.689} C_VEL
LIN {X 0,Y 751.99,Z 639.159,A -85,B 0,C 180,E1 35877.896,E2 35877.896} C_VEL
LIN {X 0,Y 753.022,Z 642.066,A -85,B 0,C 180,E1 35877.771,E2 35877.771} C_VEL
LIN {X 0,Y 755.364,Z 644.596,A -85,B 0,C 180,E1 35877.491,E2 35877.491} C_VEL
LIN {X 0,Y 755.576,Z 644.739,A -85,B 0,C 180,E1 35877.465,E2 35877.465} C_VEL
LIN {X 0,Y 755.717,Z 757.133,A -85,B 0,C 180,E1 35877.449,E2 35877.449} C_VEL
LIN {X 0,Y 756.583,Z 765.33,A -85,B 0,C 180,E1 35877.34,E2 35877.34} C_VEL
LIN {X 0,Y 757.351,Z 770.412,A -85,B 0,C 180,E1 35877.148,E2 35877.148} C_VEL
LIN {X 0,Y 757.751,Z 774.061,A -85,B 0,C 180,E1 35876.864,E2 35876.864} C_VEL
LIN {X 0,Y 757.666,Z 775.969,A -85,B 0,C 180,E1 35876.517,E2 35876.517} C_VEL
LIN {X 0,Y 757.148,Z 776.114,A -85,B 0,C 180,E1 35876.131,E2 35876.131} C_VEL
LIN {X 0,Y 756.358,Z 774.38,A -85,B 0,C 180,E1 35875.715,E2 35875.715} C_VEL
LIN {X 0,Y 755.333,Z 770.019,A -85,B 0,C 180,E1 35875.211,E2 35875.211} C_VEL
LIN {X 0,Y 754.191,Z 762.301,A -85,B 0,C 180,E1 35874.623,E2 35874.623} C_VEL
LIN {X 0,Y 753.08,Z 748.979,A -85,B 0,C 180,E1 35873.877,E2 35873.877} C_VEL
LIN {X 0,Y 752.992,Z 688.907,A -85,B 0,C 180,E1 35870.85,E2 35870.85} C_VEL
LIN {X 0,Y 753.119,Z 642.237,A -85,B 0,C 180,E1 35868.407,E2 35868.407} C_VEL
LIN {X 0,Y 751.96,Z 639.002,A -85,B 0,C 180,E1 35868.149,E2 35868.149} C_VEL
LIN {X 0,Y 751.977,Z 638.999,A -85,B 0,C 180,E1 35865.192,E2 35865.192} C_VEL
LIN {X 0,Y 751.966,Z 639.003,A -85,B 0,C 180,E1 35862.286,E2 35862.286} C_VEL
LIN {X 0,Y 751.976,Z 639.004,A -85,B 0,C 180,E1 35859.416,E2 35859.416} C_VEL
LIN {X 0,Y 751.953,Z 639.004,A -85,B 0,C 180,E1 35856.564,E2 35856.564} C_VEL
LIN {X 0,Y 751.972,Z 639,A -85,B 0,C 180,E1 35853.767,E2 35853.767} C_VEL
LIN {X 0,Y 751.974,Z 639,A -85,B 0,C 180,E1 35850.704,E2 35850.704} C_VEL
LIN {X 0,Y 751.979,Z 639.069,A -85,B 0,C 180,E1 35850.174,E2 35850.174} C_VEL
LIN {X 0,Y 752.495,Z 642.501,A -85,B 0,C 180,E1 35849.887,E2 35849.887} C_VEL
LIN {X 0,Y 752.379,Z 680.259,A -85,B 0,C 180,E1 35847.033,E2 35847.033} C_VEL
LIN {X 0,Y 752.408,Z 700.511,A -85,B 0,C 180,E1 35845.551,E2 35845.551} C_VEL
LIN {X 0,Y 752.653,Z 710.792,A -85,B 0,C 180,E1 35845.436,E2 35845.436} C_VEL
LIN {X 0,Y 752.517,Z 991.559,A -85,B 0,C 180,E1 35842.566,E2 35842.566} C_VEL
LIN {X 0,Y 752.482,Z 1013.588,A -85,B 0,C 180,E1 35842.269,E2 35842.269} C_VEL
LIN {X 0,Y 752.434,Z 1036.129,A -85,B 0,C 180,E1 35841.819,E2 35841.819} C_VEL
LIN {X 0,Y 752.392,Z 1056.779,A -85,B 0,C 180,E1 35841.273,E2 35841.273} C_VEL
LIN {X 0,Y 752.332,Z 1077.254,A -85,B 0,C 180,E1 35840.581,E2 35840.581} C_VEL
LIN {X 0,Y 752.271,Z 1097.946,A -85,B 0,C 180,E1 35839.731,E2 35839.731} C_VEL
LIN {X 0,Y 752.205,Z 1116.844,A -85,B 0,C 180,E1 35838.809,E2 35838.809} C_VEL
LIN {X 0,Y 752.154,Z 1134.974,A -85,B 0,C 180,E1 35837.764,E2 35837.764} C_VEL
LIN {X 0,Y 752.094,Z 1152.156,A -85,B 0,C 180,E1 35836.609,E2 35836.609} C_VEL
LIN {X 0,Y 752.045,Z 1168.416,A -85,B 0,C 180,E1 35835.342,E2 35835.342} C_VEL
LIN {X 0,Y 752.005,Z 1183.234,A -85,B 0,C 180,E1 35834.004,E2 35834.004} C_VEL
LIN {X 0,Y 751.975,Z 1196.704,A -85,B 0,C 180,E1 35832.581,E2 35832.581} C_VEL
LIN {X 0,Y 751.949,Z 1208.714,A -85,B 0,C 180,E1 35831.085,E2 35831.085} C_VEL
LIN {X 0,Y 751.928,Z 1219.482,A -85,B 0,C 180,E1 35829.491,E2 35829.491} C_VEL
LIN {X 0,Y 751.931,Z 1228.077,A -85,B 0,C 180,E1 35827.949,E2 35827.949} C_VEL
LIN {X 0,Y 751.913,Z 1235.19,A -85,B 0,C 180,E1 35826.337,E2 35826.337} C_VEL
LIN {X 0,Y 751.913,Z 1240.867,A -85,B 0,C 180,E1 35824.653,E2 35824.653} C_VEL
LIN {X 0,Y 751.897,Z 1244.633,A -85,B 0,C 180,E1 35823.049,E2 35823.049} C_VEL
LIN {X 0,Y 751.908,Z 1246.841,A -85,B 0,C 180,E1 35821.372,E2 35821.372} C_VEL
LIN {X 0,Y 751.915,Z 1247.409,A -85,B 0,C 180,E1 35819.619,E2 35819.619} C_VEL
LIN {X 0,Y 751.905,Z 1246.296,A -85,B 0,C 180,E1 35817.942,E2 35817.942} C_VEL
LIN {X 0,Y 751.91,Z 1243.4,A -85,B 0,C 180,E1 35816.264,E2 35816.264} C_VEL
LIN {X 0,Y 751.917,Z 1238.8,A -85,B 0,C 180,E1 35814.582,E2 35814.582} C_VEL
LIN {X 0,Y 751.915,Z 1238.521,A -85,B 0,C 180,E1 35814.498,E2 35814.498} C_VEL
LIN {X 0,Y 750.904,Z 1236.627,A -85,B 0,C 180,E1 35813.929,E2 35813.929} C_VEL
LIN {X 0,Y 744.673,Z 1230.798,A -85,B 0,C 180,E1 35812.435,E2 35812.435} C_VEL
LIN {X 0,Y 743.935,Z 1228.492,A -85,B 0,C 180,E1 35811.955,E2 35811.955} C_VEL
LIN {X 0,Y 743.946,Z 1220.017,A -85,B 0,C 180,E1 35810.406,E2 35810.406} C_VEL
LIN {X 0,Y 743.992,Z 1209.143,A -85,B 0,C 180,E1 35808.763,E2 35808.763} C_VEL
LIN {X 0,Y 744.037,Z 1197.37,A -85,B 0,C 180,E1 35807.268,E2 35807.268} C_VEL
LIN {X 0,Y 744.096,Z 1184.119,A -85,B 0,C 180,E1 35805.844,E2 35805.844} C_VEL
LIN {X 0,Y 744.181,Z 1169.467,A -85,B 0,C 180,E1 35804.492,E2 35804.492} C_VEL
LIN {X 0,Y 744.281,Z 1152.738,A -85,B 0,C 180,E1 35803.163,E2 35803.163} C_VEL
LIN {X 0,Y 744.399,Z 1135.545,A -85,B 0,C 180,E1 35801.99,E2 35801.99} C_VEL
LIN {X 0,Y 744.501,Z 1117.804,A -85,B 0,C 180,E1 35800.952,E2 35800.952} C_VEL
LIN {X 0,Y 744.631,Z 1099.114,A -85,B 0,C 180,E1 35800.021,E2 35800.021} C_VEL
LIN {X 0,Y 744.758,Z 1079.703,A -85,B 0,C 180,E1 35799.2,E2 35799.2} C_VEL
LIN {X 0,Y 744.859,Z 1059.577,A -85,B 0,C 180,E1 35798.502,E2 35798.502} C_VEL
LIN {X 0,Y 744.972,Z 1037.96,A -85,B 0,C 180,E1 35797.905,E2 35797.905} C_VEL
LIN {X 0,Y 745.054,Z 1015.94,A -85,B 0,C 180,E1 35797.445,E2 35797.445} C_VEL
LIN {X 0,Y 745.117,Z 994.274,A -85,B 0,C 180,E1 35797.138,E2 35797.138} C_VEL
LIN {X 0,Y 745.452,Z 703.204,A -85,B 0,C 180,E1 35794.131,E2 35794.131} C_VEL
LIN {X 0,Y 744.791,Z 700.055,A -85,B 0,C 180,E1 35794.066,E2 35794.066} C_VEL
LIN {X 0,Y 744.996,Z 660.844,A -85,B 0,C 180,E1 35791.107,E2 35791.107} C_VEL
LIN {X 0,Y 745.011,Z 643.666,A -85,B 0,C 180,E1 35789.782,E2 35789.782} C_VEL
LIN {X 0,Y 744.03,Z 639.993,A -85,B 0,C 180,E1 35789.425,E2 35789.425} C_VEL
LIN {X 0,Y 744.014,Z 639.987,A -85,B 0,C 180,E1 35786.564,E2 35786.564} C_VEL
LIN {X 0,Y 744.017,Z 639.993,A -85,B 0,C 180,E1 35783.741,E2 35783.741} C_VEL
LIN {X 0,Y 744.028,Z 639.986,A -85,B 0,C 180,E1 35780.844,E2 35780.844} C_VEL
LIN {X 0,Y 744.038,Z 639.983,A -85,B 0,C 180,E1 35777.887,E2 35777.887} C_VEL
LIN {X 0,Y 744.034,Z 639.991,A -85,B 0,C 180,E1 35774.873,E2 35774.873} C_VEL
LIN {X 0,Y 744.014,Z 639.986,A -85,B 0,C 180,E1 35771.996,E2 35771.996} C_VEL
LIN {X 0,Y 744.019,Z 639.988,A -85,B 0,C 180,E1 35769.271,E2 35769.271} C_VEL
LIN {X 0,Y 744.034,Z 639.987,A -85,B 0,C 180,E1 35766.391,E2 35766.391} C_VEL
LIN {X 0,Y 744.035,Z 639.982,A -85,B 0,C 180,E1 35763.343,E2 35763.343} C_VEL
LIN {X 0,Y 744.025,Z 639.987,A -85,B 0,C 180,E1 35760.352,E2 35760.352} C_VEL
LIN {X 0,Y 744.012,Z 639.989,A -85,B 0,C 180,E1 35757.537,E2 35757.537} C_VEL
LIN {X 0,Y 744.019,Z 639.985,A -85,B 0,C 180,E1 35754.703,E2 35754.703} C_VEL
LIN {X 0,Y 744.034,Z 639.992,A -85,B 0,C 180,E1 35751.772,E2 35751.772} C_VEL
LIN {X 0,Y 744.032,Z 639.984,A -85,B 0,C 180,E1 35748.817,E2 35748.817} C_VEL
LIN {X 0,Y 744.021,Z 639.985,A -85,B 0,C 180,E1 35745.832,E2 35745.832} C_VEL
LIN {X 0,Y 744.037,Z 639.992,A -85,B 0,C 180,E1 35742.891,E2 35742.891} C_VEL
LIN {X 0,Y 744.016,Z 639.985,A -85,B 0,C 180,E1 35740.063,E2 35740.063} C_VEL
LIN {X 0,Y 744.031,Z 639.986,A -85,B 0,C 180,E1 35737.181,E2 35737.181} C_VEL
LIN {X 0,Y 744.03,Z 639.989,A -85,B 0,C 180,E1 35734.24,E2 35734.24} C_VEL
LIN {X 0,Y 744.019,Z 639.984,A -85,B 0,C 180,E1 35731.31,E2 35731.31} C_VEL
LIN {X 0,Y 744.028,Z 639.989,A -85,B 0,C 180,E1 35728.461,E2 35728.461} C_VEL
LIN {X 0,Y 744.03,Z 639.985,A -85,B 0,C 180,E1 35725.608,E2 35725.608} C_VEL
LIN {X 0,Y 744.034,Z 639.982,A -85,B 0,C 180,E1 35722.652,E2 35722.652} C_VEL
LIN {X 0,Y 744.038,Z 639.989,A -85,B 0,C 180,E1 35719.627,E2 35719.627} C_VEL
LIN {X 0,Y 744.02,Z 639.986,A -85,B 0,C 180,E1 35716.716,E2 35716.716} C_VEL
LIN {X 0,Y 744.012,Z 639.987,A -85,B 0,C 180,E1 35713.849,E2 35713.849} C_VEL
LIN {X 0,Y 744.038,Z 639.99,A -85,B 0,C 180,E1 35711.023,E2 35711.023} C_VEL
LIN {X 0,Y 744.031,Z 639.983,A -85,B 0,C 180,E1 35708.064,E2 35708.064} C_VEL
LIN {X 0,Y 744.039,Z 639.984,A -85,B 0,C 180,E1 35705.042,E2 35705.042} C_VEL
LIN {X 0,Y 744.028,Z 639.991,A -85,B 0,C 180,E1 35702.118,E2 35702.118} C_VEL
LIN {X 0,Y 744.011,Z 639.986,A -85,B 0,C 180,E1 35699.292,E2 35699.292} C_VEL
LIN {X 0,Y 744.022,Z 639.992,A -85,B 0,C 180,E1 35696.474,E2 35696.474} C_VEL
LIN {X 0,Y 744.031,Z 639.984,A -85,B 0,C 180,E1 35693.561,E2 35693.561} C_VEL
LIN {X 0,Y 744.038,Z 639.982,A -85,B 0,C 180,E1 35690.478,E2 35690.478} C_VEL
LIN {X 0,Y 744.03,Z 639.989,A -85,B 0,C 180,E1 35687.43,E2 35687.43} C_VEL
LIN {X 0,Y 744.014,Z 639.989,A -85,B 0,C 180,E1 35684.582,E2 35684.582} C_VEL
LIN {X 0,Y 744.014,Z 639.988,A -85,B 0,C 180,E1 35681.769,E2 35681.769} C_VEL
LIN {X 0,Y 744.038,Z 639.989,A -85,B 0,C 180,E1 35678.873,E2 35678.873} C_VEL
LIN {X 0,Y 744.06,Z 640.157,A -85,B 0,C 180,E1 35678.772,E2 35678.772} C_VEL
LIN {X 0,Y 745.346,Z 644.756,A -85,B 0,C 180,E1 35678.398,E2 35678.398} C_VEL
LIN {X 0,Y 745.155,Z 689.298,A -85,B 0,C 180,E1 35675.428,E2 35675.428} C_VEL
LIN {X 0,Y 744.663,Z 732.034,A -85,B 0,C 180,E1 35672.623,E2 35672.623} C_VEL
LIN {X 0,Y 744.496,Z 777.051,A -85,B 0,C 180,E1 35669.797,E2 35669.797} C_VEL
LIN {X 0,Y 744.335,Z 823.788,A -85,B 0,C 180,E1 35666.917,E2 35666.917} C_VEL
LIN {X 0,Y 744.189,Z 871.457,A -85,B 0,C 180,E1 35664.024,E2 35664.024} C_VEL
LIN {X 0,Y 744.201,Z 891.684,A -85,B 0,C 180,E1 35662.827,E2 35662.827} C_VEL
LIN {X 0,Y 744.212,Z 1033.468,A -85,B 0,C 180,E1 35661.435,E2 35661.435} C_VEL
LIN {X 0,Y 744.184,Z 1050.303,A -85,B 0,C 180,E1 35661.121,E2 35661.121} C_VEL
LIN {X 0,Y 744.132,Z 1066.468,A -85,B 0,C 180,E1 35660.659,E2 35660.659} C_VEL
LIN {X 0,Y 744.079,Z 1080.381,A -85,B 0,C 180,E1 35660.122,E2 35660.122} C_VEL
LIN {X 0,Y 744.062,Z 1093.689,A -85,B 0,C 180,E1 35659.467,E2 35659.467} C_VEL
LIN {X 0,Y 744.026,Z 1105.724,A -85,B 0,C 180,E1 35658.735,E2 35658.735} C_VEL
LIN {X 0,Y 743.99,Z 1118.486,A -85,B 0,C 180,E1 35657.763,E2 35657.763} C_VEL
LIN {X 0,Y 743.952,Z 1128.598,A -85,B 0,C 180,E1 35656.796,E2 35656.796} C_VEL
LIN {X 0,Y 743.935,Z 1137.33,A -85,B 0,C 180,E1 35655.754,E2 35655.754} C_VEL
LIN {X 0,Y 743.925,Z 1144.677,A -85,B 0,C 180,E1 35654.637,E2 35654.637} C_VEL
LIN {X 0,Y 743.918,Z 1150.504,A -85,B 0,C 180,E1 35653.446,E2 35653.446} C_VEL
LIN {X 0,Y 743.916,Z 1154.671,A -85,B 0,C 180,E1 35652.182,E2 35652.182} C_VEL
LIN {X 0,Y 743.918,Z 1156.853,A -85,B 0,C 180,E1 35651.003,E2 35651.003} C_VEL
LIN {X 0,Y 743.915,Z 1157.448,A -85,B 0,C 180,E1 35649.75,E2 35649.75} C_VEL
LIN {X 0,Y 743.915,Z 1156.177,A -85,B 0,C 180,E1 35648.422,E2 35648.422} C_VEL
LIN {X 0,Y 743.916,Z 1153.093,A -85,B 0,C 180,E1 35647.181,E2 35647.181} C_VEL
LIN {X 0,Y 743.919,Z 1148.274,A -85,B 0,C 180,E1 35645.964,E2 35645.964} C_VEL
LIN {X 0,Y 743.928,Z 1142.182,A -85,B 0,C 180,E1 35644.857,E2 35644.857} C_VEL
LIN {X 0,Y 743.944,Z 1133.771,A -85,B 0,C 180,E1 35643.699,E2 35643.699} C_VEL
LIN {X 0,Y 743.972,Z 1123.693,A -85,B 0,C 180,E1 35642.619,E2 35642.619} C_VEL
LIN {X 0,Y 744.001,Z 1112.856,A -85,B 0,C 180,E1 35641.694,E2 35641.694} C_VEL
LIN {X 0,Y 744.036,Z 1101.246,A -85,B 0,C 180,E1 35640.886,E2 35640.886} C_VEL
LIN {X 0,Y 744.066,Z 1088.27,A -85,B 0,C 180,E1 35640.154,E2 35640.154} C_VEL
LIN {X 0,Y 744.117,Z 1072.402,A -85,B 0,C 180,E1 35639.461,E2 35639.461} C_VEL
LIN {X 0,Y 744.167,Z 1057.643,A -85,B 0,C 180,E1 35638.98,E2 35638.98} C_VEL
LIN {X 0,Y 744.191,Z 1042.106,A -85,B 0,C 180,E1 35638.617,E2 35638.617} C_VEL
LIN {X 0,Y 744.222,Z 1024.957,A -85,B 0,C 180,E1 35638.372,E2 35638.372} C_VEL
LIN {X 0,Y 744.158,Z 891.176,A -85,B 0,C 180,E1 35637.073,E2 35637.073} C_VEL
LIN {X 0,Y 744.286,Z 842.605,A -85,B 0,C 180,E1 35634.14,E2 35634.14} C_VEL
LIN {X 0,Y 744.418,Z 795.112,A -85,B 0,C 180,E1 35631.231,E2 35631.231} C_VEL
LIN {X 0,Y 744.58,Z 750.552,A -85,B 0,C 180,E1 35628.458,E2 35628.458} C_VEL
LIN {X 0,Y 744.783,Z 731.846,A -85,B 0,C 180,E1 35627.241,E2 35627.241} C_VEL
LIN {X 0,Y 745.911,Z 691.986,A -85,B 0,C 180,E1 35624.489,E2 35624.489} C_VEL
LIN {X 0,Y 746.169,Z 653.311,A -85,B 0,C 180,E1 35621.685,E2 35621.685} C_VEL
LIN {X 0,Y 746.063,Z 645.734,A -85,B 0,C 180,E1 35621.114,E2 35621.114} C_VEL
LIN {X 0,Y 744.028,Z 639.994,A -85,B 0,C 180,E1 35620.532,E2 35620.532} C_VEL
LIN {X 0,Y 744.032,Z 639.981,A -85,B 0,C 180,E1 35617.563,E2 35617.563} C_VEL
LIN {X 0,Y 744.033,Z 639.993,A -85,B 0,C 180,E1 35614.53,E2 35614.53} C_VEL
LIN {X 0,Y 744.031,Z 639.981,A -85,B 0,C 180,E1 35611.505,E2 35611.505} C_VEL
LIN {X 0,Y 744.018,Z 639.99,A -85,B 0,C 180,E1 35608.571,E2 35608.571} C_VEL
LIN {X 0,Y 744.012,Z 639.987,A -85,B 0,C 180,E1 35605.738,E2 35605.738} C_VEL
LIN {X 0,Y 744.026,Z 639.982,A -85,B 0,C 180,E1 35602.885,E2 35602.885} C_VEL
LIN {X 0,Y 744.039,Z 639.992,A -85,B 0,C 180,E1 35599.93,E2 35599.93} C_VEL
LIN {X 0,Y 744.027,Z 639.982,A -85,B 0,C 180,E1 35596.945,E2 35596.945} C_VEL
LIN {X 0,Y 744.025,Z 639.992,A -85,B 0,C 180,E1 35594.008,E2 35594.008} C_VEL
LIN {X 0,Y 744.049,Z 640.092,A -85,B 0,C 180,E1 35591.733,E2 35591.733} C_VEL
LIN {X 0,Y 745.796,Z 645.382,A -85,B 0,C 180,E1 35591.371,E2 35591.371} C_VEL
LIN {X 0,Y 745.42,Z 696.387,A -85,B 0,C 180,E1 35588.883,E2 35588.883} C_VEL
LIN {X 0,Y 745.676,Z 750.937,A -85,B 0,C 180,E1 35586.303,E2 35586.303} C_VEL
LIN {X 0,Y 747.613,Z 767.153,A -85,B 0,C 180,E1 35585.48,E2 35585.48} C_VEL
LIN {X 0,Y 749.684,Z 775.325,A -85,B 0,C 180,E1 35584.956,E2 35584.956} C_VEL
LIN {X 0,Y 751.794,Z 780.577,A -85,B 0,C 180,E1 35584.451,E2 35584.451} C_VEL
LIN {X 0,Y 753.637,Z 783.179,A -85,B 0,C 180,E1 35583.981,E2 35583.981} C_VEL
LIN {X 0,Y 754.882,Z 783.744,A -85,B 0,C 180,E1 35583.576,E2 35583.576} C_VEL
LIN {X 0,Y 755.601,Z 782.711,A -85,B 0,C 180,E1 35583.15,E2 35583.15} C_VEL
LIN {X 0,Y 755.498,Z 779.949,A -85,B 0,C 180,E1 35582.759,E2 35582.759} C_VEL
LIN {X 0,Y 754.592,Z 775.865,A -85,B 0,C 180,E1 35582.454,E2 35582.454} C_VEL
LIN {X 0,Y 753.007,Z 770.041,A -85,B 0,C 180,E1 35582.227,E2 35582.227} C_VEL
LIN {X 0,Y 751.744,Z 761.894,A -85,B 0,C 180,E1 35582.074,E2 35582.074} C_VEL
LIN {X 0,Y 751.312,Z 752.352,A -85,B 0,C 180,E1 35582.021,E2 35582.021} C_VEL
LIN {X 0,Y 751.258,Z 649.602,A -85,B 0,C 180,E1 35582.015,E2 35582.015} C_VEL
LIN {X 0,Y 749.232,Z 646.522,A -85,B 0,C 180,E1 35581.766,E2 35581.766} C_VEL
LIN {X 0,Y 745.62,Z 644.842,A -85,B 0,C 180,E1 35581.307,E2 35581.307} C_VEL
LIN {X 0,Y 745.364,Z 700.186,A -85,B 0,C 180,E1 35578.612,E2 35578.612} C_VEL
LIN {X 0,Y 745.142,Z 757.721,A -85,B 0,C 180,E1 35575.893,E2 35575.893} C_VEL
LIN {X 0,Y 745.432,Z 765.893,A -85,B 0,C 180,E1 35575.797,E2 35575.797} C_VEL
LIN {X 0,Y 745.145,Z 1033.446,A -85,B 0,C 180,E1 35573.033,E2 35573.033} C_VEL
LIN {X 0,Y 745.076,Z 1066.841,A -85,B 0,C 180,E1 35572.657,E2 35572.657} C_VEL
LIN {X 0,Y 745.02,Z 1088.956,A -85,B 0,C 180,E1 35572.258,E2 35572.258} C_VEL
LIN {X 0,Y 744.906,Z 1109.914,A -85,B 0,C 180,E1 35571.739,E2 35571.739} C_VEL
LIN {X 0,Y 744.792,Z 1130.742,A -85,B 0,C 180,E1 35571.085,E2 35571.085} C_VEL
LIN {X 0,Y 744.697,Z 1150.755,A -85,B 0,C 180,E1 35570.308,E2 35570.308} C_VEL
LIN {X 0,Y 744.557,Z 1170.766,A -85,B 0,C 180,E1 35569.371,E2 35569.371} C_VEL
LIN {X 0,Y 744.421,Z 1189.813,A -85,B 0,C 180,E1 35568.317,E2 35568.317} C_VEL
LIN {X 0,Y 744.321,Z 1207.255,A -85,B 0,C 180,E1 35567.188,E2 35567.188} C_VEL
LIN {X 0,Y 744.223,Z 1223.722,A -85,B 0,C 180,E1 35565.946,E2 35565.946} C_VEL
LIN {X 0,Y 744.127,Z 1238.732,A -85,B 0,C 180,E1 35564.631,E2 35564.631} C_VEL
LIN {X 0,Y 744.046,Z 1252.761,A -85,B 0,C 180,E1 35563.205,E2 35563.205} C_VEL
LIN {X 0,Y 744.004,Z 1265.349,A -85,B 0,C 180,E1 35561.707,E2 35561.707} C_VEL
LIN {X 0,Y 743.956,Z 1275.852,A -85,B 0,C 180,E1 35560.218,E2 35560.218} C_VEL
LIN {X 0,Y 743.929,Z 1285.488,A -85,B 0,C 180,E1 35558.579,E2 35558.579} C_VEL
LIN {X 0,Y 743.916,Z 1293.247,A -85,B 0,C 180,E1 35556.947,E2 35556.947} C_VEL
LIN {X 0,Y 743.921,Z 1299.157,A -85,B 0,C 180,E1 35555.32,E2 35555.32} C_VEL
LIN {X 0,Y 743.914,Z 1303.631,A -85,B 0,C 180,E1 35553.621,E2 35553.621} C_VEL
LIN {X 0,Y 743.911,Z 1306.412,A -85,B 0,C 180,E1 35551.925,E2 35551.925} C_VEL
LIN {X 0,Y 743.899,Z 1307.418,A -85,B 0,C 180,E1 35550.307,E2 35550.307} C_VEL
LIN {X 0,Y 743.904,Z 1306.885,A -85,B 0,C 180,E1 35548.613,E2 35548.613} C_VEL
LIN {X 0,Y 743.917,Z 1304.727,A -85,B 0,C 180,E1 35546.917,E2 35546.917} C_VEL
LIN {X 0,Y 743.906,Z 1300.784,A -85,B 0,C 180,E1 35545.219,E2 35545.219} C_VEL
LIN {X 0,Y 743.912,Z 1295.064,A -85,B 0,C 180,E1 35543.516,E2 35543.516} C_VEL
LIN {X 0,Y 743.935,Z 1287.914,A -85,B 0,C 180,E1 35541.886,E2 35541.886} C_VEL
LIN {X 0,Y 743.955,Z 1278.831,A -85,B 0,C 180,E1 35540.249,E2 35540.249} C_VEL
LIN {X 0,Y 743.992,Z 1268.219,A -85,B 0,C 180,E1 35538.683,E2 35538.683} C_VEL
LIN {X 0,Y 744.046,Z 1256.269,A -85,B 0,C 180,E1 35537.188,E2 35537.188} C_VEL
LIN {X 0,Y 744.114,Z 1242.896,A -85,B 0,C 180,E1 35535.764,E2 35535.764} C_VEL
LIN {X 0,Y 744.185,Z 1228.002,A -85,B 0,C 180,E1 35534.411,E2 35534.411} C_VEL
LIN {X 0,Y 744.285,Z 1211.129,A -85,B 0,C 180,E1 35533.09,E2 35533.09} C_VEL
LIN {X 0,Y 744.414,Z 1192.849,A -85,B 0,C 180,E1 35531.869,E2 35531.869} C_VEL
LIN {X 0,Y 744.541,Z 1174.717,A -85,B 0,C 180,E1 35530.83,E2 35530.83} C_VEL
LIN {X 0,Y 744.651,Z 1155.385,A -85,B 0,C 180,E1 35529.894,E2 35529.894} C_VEL
LIN {X 0,Y 744.769,Z 1135.131,A -85,B 0,C 180,E1 35529.076,E2 35529.076} C_VEL
LIN {X 0,Y 744.899,Z 1114.09,A -85,B 0,C 180,E1 35528.378,E2 35528.378} C_VEL
LIN {X 0,Y 744.988,Z 1092.686,A -85,B 0,C 180,E1 35527.824,E2 35527.824} C_VEL
LIN {X 0,Y 745.069,Z 1070.906,A -85,B 0,C 180,E1 35527.408,E2 35527.408} C_VEL
LIN {X 0,Y 745.129,Z 1046.999,A -85,B 0,C 180,E1 35527.105,E2 35527.105} C_VEL
LIN {X 0,Y 745.426,Z 776.106,A -85,B 0,C 180,E1 35524.31,E2 35524.31} C_VEL
LIN {X 0,Y 745.205,Z 758.138,A -85,B 0,C 180,E1 35524.113,E2 35524.113} C_VEL
LIN {X 0,Y 745.101,Z 754.573,A -85,B 0,C 180,E1 35523.971,E2 35523.971} C_VEL
LIN {X 0,Y 745.366,Z 697.415,A -85,B 0,C 180,E1 35521.254,E2 35521.254} C_VEL
LIN {X 0,Y 745.65,Z 644.701,A -85,B 0,C 180,E1 35518.681,E2 35518.681} C_VEL
LIN {X 0,Y 749.576,Z 646.873,A -85,B 0,C 180,E1 35518.191,E2 35518.191} C_VEL
LIN {X 0,Y 751.305,Z 649.66,A -85,B 0,C 180,E1 35517.98,E2 35517.98} C_VEL
LIN {X 0,Y 751.444,Z 757.496,A -85,B 0,C 180,E1 35517.963,E2 35517.963} C_VEL
LIN {X 0,Y 752.356,Z 766.734,A -85,B 0,C 180,E1 35517.852,E2 35517.852} C_VEL
LIN {X 0,Y 754.018,Z 773.817,A -85,B 0,C 180,E1 35517.646,E2 35517.646} C_VEL
LIN {X 0,Y 755.23,Z 778.491,A -85,B 0,C 180,E1 35517.371,E2 35517.371} C_VEL
LIN {X 0,Y 755.672,Z 781.707,A -85,B 0,C 180,E1 35517.024,E2 35517.024} C_VEL
LIN {X 0,Y 755.344,Z 783.434,A -85,B 0,C 180,E1 35516.646,E2 35516.646} C_VEL
LIN {X 0,Y 754.297,Z 783.648,A -85,B 0,C 180,E1 35516.217,E2 35516.217} C_VEL
LIN {X 0,Y 752.896,Z 782.346,A -85,B 0,C 180,E1 35515.821,E2 35515.821} C_VEL
LIN {X 0,Y 750.981,Z 778.82,A -85,B 0,C 180,E1 35515.352,E2 35515.352} C_VEL
LIN {X 0,Y 748.979,Z 772.962,A -85,B 0,C 180,E1 35514.873,E2 35514.873} C_VEL
LIN {X 0,Y 746.98,Z 762.906,A -85,B 0,C 180,E1 35514.277,E2 35514.277} C_VEL
LIN {X 0,Y 745.817,Z 745.759,A -85,B 0,C 180,E1 35513.373,E2 35513.373} C_VEL
LIN {X 0,Y 746.089,Z 692.258,A -85,B 0,C 180,E1 35510.65,E2 35510.65} C_VEL
LIN {X 0,Y 746.377,Z 646.06,A -85,B 0,C 180,E1 35508.21,E2 35508.21} C_VEL
LIN {X 0,Y 744.015,Z 640.009,A -85,B 0,C 180,E1 35507.737,E2 35507.737} C_VEL
LIN {X 0,Y 744.039,Z 639.989,A -85,B 0,C 180,E1 35504.873,E2 35504.873} C_VEL
LIN {X 0,Y 744.03,Z 639.993,A -85,B 0,C 180,E1 35501.998,E2 35501.998} C_VEL
LIN {X 0,Y 744.039,Z 639.988,A -85,B 0,C 180,E1 35499.035,E2 35499.035} C_VEL
LIN {X 0,Y 744.033,Z 639.989,A -85,B 0,C 180,E1 35495.964,E2 35495.964} C_VEL
LIN {X 0,Y 744.025,Z 639.993,A -85,B 0,C 180,E1 35493.008,E2 35493.008} C_VEL
LIN {X 0,Y 744.068,Z 640.221,A -85,B 0,C 180,E1 35490.439,E2 35490.439} C_VEL
LIN {X 0,Y 745.085,Z 644.797,A -85,B 0,C 180,E1 35490.037,E2 35490.037} C_VEL
LIN {X 0,Y 744.865,Z 682.555,A -85,B 0,C 180,E1 35487.156,E2 35487.156} C_VEL
LIN {X 0,Y 744.87,Z 700.585,A -85,B 0,C 180,E1 35485.828,E2 35485.828} C_VEL
LIN {X 0,Y 745.438,Z 704.681,A -85,B 0,C 180,E1 35485.764,E2 35485.764} C_VEL
LIN {X 0,Y 745.133,Z 988.516,A -85,B 0,C 180,E1 35482.834,E2 35482.834} C_VEL
LIN {X 0,Y 745.069,Z 1012.018,A -85,B 0,C 180,E1 35482.529,E2 35482.529} C_VEL
LIN {X 0,Y 744.978,Z 1034.221,A -85,B 0,C 180,E1 35482.095,E2 35482.095} C_VEL
LIN {X 0,Y 744.894,Z 1054.851,A -85,B 0,C 180,E1 35481.554,E2 35481.554} C_VEL
LIN {X 0,Y 744.767,Z 1075.495,A -85,B 0,C 180,E1 35480.865,E2 35480.865} C_VEL
LIN {X 0,Y 744.641,Z 1096.179,A -85,B 0,C 180,E1 35480.024,E2 35480.024} C_VEL
LIN {X 0,Y 744.54,Z 1115.438,A -85,B 0,C 180,E1 35479.088,E2 35479.088} C_VEL
LIN {X 0,Y 744.405,Z 1134.052,A -85,B 0,C 180,E1 35478.012,E2 35478.012} C_VEL
LIN {X 0,Y 744.282,Z 1151.494,A -85,B 0,C 180,E1 35476.837,E2 35476.837} C_VEL
LIN {X 0,Y 744.182,Z 1167.874,A -85,B 0,C 180,E1 35475.556,E2 35475.556} C_VEL
LIN {X 0,Y 744.116,Z 1182.455,A -85,B 0,C 180,E1 35474.235,E2 35474.235} C_VEL
LIN {X 0,Y 744.048,Z 1195.87,A -85,B 0,C 180,E1 35472.811,E2 35472.811} C_VEL
LIN {X 0,Y 743.99,Z 1207.905,A -85,B 0,C 180,E1 35471.316,E2 35471.316} C_VEL
LIN {X 0,Y 743.965,Z 1218.103,A -85,B 0,C 180,E1 35469.828,E2 35469.828} C_VEL
LIN {X 0,Y 743.925,Z 1226.863,A -85,B 0,C 180,E1 35468.269,E2 35468.269} C_VEL
LIN {X 0,Y 743.912,Z 1234.587,A -85,B 0,C 180,E1 35466.56,E2 35466.56} C_VEL
LIN {X 0,Y 743.903,Z 1240.253,A -85,B 0,C 180,E1 35464.935,E2 35464.935} C_VEL
LIN {X 0,Y 743.903,Z 1244.161,A -85,B 0,C 180,E1 35463.313,E2 35463.313} C_VEL
LIN {X 0,Y 743.915,Z 1246.709,A -85,B 0,C 180,E1 35461.54,E2 35461.54} C_VEL
LIN {X 0,Y 743.915,Z 1247.475,A -85,B 0,C 180,E1 35459.846,E2 35459.846} C_VEL
LIN {X 0,Y 743.916,Z 1246.521,A -85,B 0,C 180,E1 35458.151,E2 35458.151} C_VEL
LIN {X 0,Y 743.911,Z 1243.872,A -85,B 0,C 180,E1 35456.455,E2 35456.455} C_VEL
LIN {X 0,Y 743.912,Z 1239.557,A -85,B 0,C 180,E1 35454.756,E2 35454.756} C_VEL
LIN {X 0,Y 743.926,Z 1233.728,A -85,B 0,C 180,E1 35453.13,E2 35453.13} C_VEL
LIN {X 0,Y 743.935,Z 1228.492,A -85,B 0,C 180,E1 35451.955,E2 35451.955} C_VEL
LIN {X 0,Y 742.949,Z 1225.686,A -85,B 0,C 180,E1 35451.403,E2 35451.403} C_VEL
LIN {X 0,Y 736.724,Z 1217.891,A -85,B 0,C 180,E1 35449.949,E2 35449.949} C_VEL
LIN {X 0,Y 735.996,Z 1214.931,A -85,B 0,C 180,E1 35449.485,E2 35449.485} C_VEL
LIN {X 0,Y 736.068,Z 1203.822,A -85,B 0,C 180,E1 35447.925,E2 35447.925} C_VEL
LIN {X 0,Y 736.155,Z 1191.026,A -85,B 0,C 180,E1 35446.41,E2 35446.41} C_VEL
LIN {X 0,Y 736.25,Z 1177.491,A -85,B 0,C 180,E1 35445.046,E2 35445.046} C_VEL
LIN {X 0,Y 736.391,Z 1161.233,A -85,B 0,C 180,E1 35443.635,E2 35443.635} C_VEL
LIN {X 0,Y 736.561,Z 1144.336,A -85,B 0,C 180,E1 35442.379,E2 35442.379} C_VEL
LIN {X 0,Y 736.751,Z 1126.509,A -85,B 0,C 180,E1 35441.237,E2 35441.237} C_VEL
LIN {X 0,Y 736.914,Z 1107.578,A -85,B 0,C 180,E1 35440.212,E2 35440.212} C_VEL
LIN {X 0,Y 737.113,Z 1088.02,A -85,B 0,C 180,E1 35439.316,E2 35439.316} C_VEL
LIN {X 0,Y 737.291,Z 1068.437,A -85,B 0,C 180,E1 35438.562,E2 35438.562} C_VEL
LIN {X 0,Y 737.441,Z 1047.59,A -85,B 0,C 180,E1 35437.919,E2 35437.919} C_VEL
LIN {X 0,Y 737.599,Z 1025.304,A -85,B 0,C 180,E1 35437.386,E2 35437.386} C_VEL
LIN {X 0,Y 737.713,Z 1003.103,A -85,B 0,C 180,E1 35437.006,E2 35437.006} C_VEL
LIN {X 0,Y 737.941,Z 865.001,A -85,B 0,C 180,E1 35435.554,E2 35435.554} C_VEL
LIN {X 0,Y 738.037,Z 703.686,A -85,B 0,C 180,E1 35433.857,E2 35433.857} C_VEL
LIN {X 0,Y 737.249,Z 700.02,A -85,B 0,C 180,E1 35433.778,E2 35433.778} C_VEL
LIN {X 0,Y 737.555,Z 661.981,A -85,B 0,C 180,E1 35430.877,E2 35430.877} C_VEL
LIN {X 0,Y 737.505,Z 645.949,A -85,B 0,C 180,E1 35429.622,E2 35429.622} C_VEL
LIN {X 0,Y 736.092,Z 640.981,A -85,B 0,C 180,E1 35429.148,E2 35429.148} C_VEL
LIN {X 0,Y 736.093,Z 640.976,A -85,B 0,C 180,E1 35426.235,E2 35426.235} C_VEL
LIN {X 0,Y 736.089,Z 640.974,A -85,B 0,C 180,E1 35423.198,E2 35423.198} C_VEL
LIN {X 0,Y 736.101,Z 640.979,A -85,B 0,C 180,E1 35420.224,E2 35420.224} C_VEL
LIN {X 0,Y 736.073,Z 640.977,A -85,B 0,C 180,E1 35417.299,E2 35417.299} C_VEL
LIN {X 0,Y 736.082,Z 640.976,A -85,B 0,C 180,E1 35414.502,E2 35414.502} C_VEL
LIN {X 0,Y 736.103,Z 640.979,A -85,B 0,C 180,E1 35411.543,E2 35411.543} C_VEL
LIN {X 0,Y 736.1,Z 640.973,A -85,B 0,C 180,E1 35408.472,E2 35408.472} C_VEL
LIN {X 0,Y 736.099,Z 640.972,A -85,B 0,C 180,E1 35405.357,E2 35405.357} C_VEL
LIN {X 0,Y 736.096,Z 640.977,A -85,B 0,C 180,E1 35402.266,E2 35402.266} C_VEL
LIN {X 0,Y 736.082,Z 640.976,A -85,B 0,C 180,E1 35399.366,E2 35399.366} C_VEL
LIN {X 0,Y 736.074,Z 640.974,A -85,B 0,C 180,E1 35396.46,E2 35396.46} C_VEL
LIN {X 0,Y 736.096,Z 640.982,A -85,B 0,C 180,E1 35393.624,E2 35393.624} C_VEL
LIN {X 0,Y 736.093,Z 640.973,A -85,B 0,C 180,E1 35390.622,E2 35390.622} C_VEL
LIN {X 0,Y 736.095,Z 640.972,A -85,B 0,C 180,E1 35387.634,E2 35387.634} C_VEL
LIN {X 0,Y 736.098,Z 640.978,A -85,B 0,C 180,E1 35384.555,E2 35384.555} C_VEL
LIN {X 0,Y 736.088,Z 640.975,A -85,B 0,C 180,E1 35381.599,E2 35381.599} C_VEL
LIN {X 0,Y 736.076,Z 640.973,A -85,B 0,C 180,E1 35378.673,E2 35378.673} C_VEL
LIN {X 0,Y 736.097,Z 640.981,A -85,B 0,C 180,E1 35375.848,E2 35375.848} C_VEL
LIN {X 0,Y 736.082,Z 640.974,A -85,B 0,C 180,E1 35372.882,E2 35372.882} C_VEL
LIN {X 0,Y 736.095,Z 640.972,A -85,B 0,C 180,E1 35369.923,E2 35369.923} C_VEL
LIN {X 0,Y 736.094,Z 640.981,A -85,B 0,C 180,E1 35366.964,E2 35366.964} C_VEL
LIN {X 0,Y 736.082,Z 640.974,A -85,B 0,C 180,E1 35363.997,E2 35363.997} C_VEL
LIN {X 0,Y 736.073,Z 640.978,A -85,B 0,C 180,E1 35361.171,E2 35361.171} C_VEL
LIN {X 0,Y 736.083,Z 640.977,A -85,B 0,C 180,E1 35358.324,E2 35358.324} C_VEL
LIN {X 0,Y 736.095,Z 640.971,A -85,B 0,C 180,E1 35355.367,E2 35355.367} C_VEL
LIN {X 0,Y 736.097,Z 640.975,A -85,B 0,C 180,E1 35352.287,E2 35352.287} C_VEL
LIN {X 0,Y 736.09,Z 640.978,A -85,B 0,C 180,E1 35349.32,E2 35349.32} C_VEL
LIN {X 0,Y 736.077,Z 640.974,A -85,B 0,C 180,E1 35346.378,E2 35346.378} C_VEL
LIN {X 0,Y 736.09,Z 640.978,A -85,B 0,C 180,E1 35343.531,E2 35343.531} C_VEL
LIN {X 0,Y 736.092,Z 640.975,A -85,B 0,C 180,E1 35340.637,E2 35340.637} C_VEL
LIN {X 0,Y 736.091,Z 640.971,A -85,B 0,C 180,E1 35337.644,E2 35337.644} C_VEL
LIN {X 0,Y 736.098,Z 640.976,A -85,B 0,C 180,E1 35334.59,E2 35334.59} C_VEL
LIN {X 0,Y 736.084,Z 640.977,A -85,B 0,C 180,E1 35331.728,E2 35331.728} C_VEL
LIN {X 0,Y 736.073,Z 640.975,A -85,B 0,C 180,E1 35328.895,E2 35328.895} C_VEL
LIN {X 0,Y 736.101,Z 640.98,A -85,B 0,C 180,E1 35326.045,E2 35326.045} C_VEL
LIN {X 0,Y 736.088,Z 640.974,A -85,B 0,C 180,E1 35323.048,E2 35323.048} C_VEL
LIN {X 0,Y 736.097,Z 640.977,A -85,B 0,C 180,E1 35319.996,E2 35319.996} C_VEL
LIN {X 0,Y 736.125,Z 641.194,A -85,B 0,C 180,E1 35319.082,E2 35319.082} C_VEL
LIN {X 0,Y 738.076,Z 647.608,A -85,B 0,C 180,E1 35318.548,E2 35318.548} C_VEL
LIN {X 0,Y 737.777,Z 693.046,A -85,B 0,C 180,E1 35315.498,E2 35315.498} C_VEL
LIN {X 0,Y 737.16,Z 736.563,A -85,B 0,C 180,E1 35312.617,E2 35312.617} C_VEL
LIN {X 0,Y 736.81,Z 777.174,A -85,B 0,C 180,E1 35310.005,E2 35310.005} C_VEL
LIN {X 0,Y 736.556,Z 824.404,A -85,B 0,C 180,E1 35307.064,E2 35307.064} C_VEL
LIN {X 0,Y 736.348,Z 870.901,A -85,B 0,C 180,E1 35304.21,E2 35304.21} C_VEL
LIN {X 0,Y 736.335,Z 891.742,A -85,B 0,C 180,E1 35302.966,E2 35302.966} C_VEL
LIN {X 0,Y 736.367,Z 1033.149,A -85,B 0,C 180,E1 35301.562,E2 35301.562} C_VEL
LIN {X 0,Y 736.328,Z 1049.138,A -85,B 0,C 180,E1 35301.269,E2 35301.269} C_VEL
LIN {X 0,Y 736.257,Z 1065.809,A -85,B 0,C 180,E1 35300.798,E2 35300.798} C_VEL
LIN {X 0,Y 736.181,Z 1079.643,A -85,B 0,C 180,E1 35300.264,E2 35300.264} C_VEL
LIN {X 0,Y 736.131,Z 1092.145,A -85,B 0,C 180,E1 35299.654,E2 35299.654} C_VEL
LIN {X 0,Y 736.087,Z 1103.958,A -85,B 0,C 180,E1 35298.945,E2 35298.945} C_VEL
LIN {X 0,Y 736.039,Z 1114.588,A -85,B 0,C 180,E1 35298.166,E2 35298.166} C_VEL
LIN {X 0,Y 735.993,Z 1125.176,A -85,B 0,C 180,E1 35297.228,E2 35297.228} C_VEL
LIN {X 0,Y 735.954,Z 1135.283,A -85,B 0,C 180,E1 35296.091,E2 35296.091} C_VEL
LIN {X 0,Y 735.935,Z 1142.886,A -85,B 0,C 180,E1 35294.989,E2 35294.989} C_VEL
LIN {X 0,Y 735.921,Z 1148.975,A -85,B 0,C 180,E1 35293.835,E2 35293.835} C_VEL
LIN {X 0,Y 735.919,Z 1153.746,A -85,B 0,C 180,E1 35292.556,E2 35292.556} C_VEL
LIN {X 0,Y 735.917,Z 1156.614,A -85,B 0,C 180,E1 35291.203,E2 35291.203} C_VEL
LIN {X 0,Y 735.916,Z 1157.458,A -85,B 0,C 180,E1 35290.016,E2 35290.016} C_VEL
LIN {X 0,Y 735.918,Z 1156.768,A -85,B 0,C 180,E1 35288.832,E2 35288.832} C_VEL
LIN {X 0,Y 735.916,Z 1154.332,A -85,B 0,C 180,E1 35287.573,E2 35287.573} C_VEL
LIN {X 0,Y 735.922,Z 1149.721,A -85,B 0,C 180,E1 35286.24,E2 35286.24} C_VEL
LIN {X 0,Y 735.932,Z 1143.756,A -85,B 0,C 180,E1 35285.067,E2 35285.067} C_VEL
LIN {X 0,Y 735.948,Z 1136.429,A -85,B 0,C 180,E1 35283.973,E2 35283.973} C_VEL
LIN {X 0,Y 735.982,Z 1127.864,A -85,B 0,C 180,E1 35282.959,E2 35282.959} C_VEL
LIN {X 0,Y 736.03,Z 1117.077,A -85,B 0,C 180,E1 35281.946,E2 35281.946} C_VEL
LIN {X 0,Y 736.083,Z 1105.269,A -85,B 0,C 180,E1 35281.051,E2 35281.051} C_VEL
LIN {X 0,Y 736.138,Z 1093.158,A -85,B 0,C 180,E1 35280.311,E2 35280.311} C_VEL
LIN {X 0,Y 736.171,Z 1080.604,A -85,B 0,C 180,E1 35279.689,E2 35279.689} C_VEL
LIN {X 0,Y 736.258,Z 1066.718,A -85,B 0,C 180,E1 35279.144,E2 35279.144} C_VEL
LIN {X 0,Y 736.322,Z 1050.389,A -85,B 0,C 180,E1 35278.67,E2 35278.67} C_VEL
LIN {X 0,Y 736.359,Z 1033.796,A -85,B 0,C 180,E1 35278.356,E2 35278.356} C_VEL
LIN {X 0,Y 736.412,Z 972.051,A -85,B 0,C 180,E1 35277.731,E2 35277.731} C_VEL
LIN {X 0,Y 736.285,Z 891.204,A -85,B 0,C 180,E1 35276.935,E2 35276.935} C_VEL
LIN {X 0,Y 736.481,Z 843.118,A -85,B 0,C 180,E1 35273.999,E2 35273.999} C_VEL
LIN {X 0,Y 736.697,Z 794.999,A -85,B 0,C 180,E1 35271.02,E2 35271.02} C_VEL
LIN {X 0,Y 736.964,Z 761.516,A -85,B 0,C 180,E1 35268.892,E2 35268.892} C_VEL
LIN {X 0,Y 738.121,Z 720.095,A -85,B 0,C 180,E1 35266.047,E2 35266.047} C_VEL
LIN {X 0,Y 738.962,Z 690.065,A -85,B 0,C 180,E1 35263.936,E2 35263.936} C_VEL
LIN {X 0,Y 739.44,Z 651.547,A -85,B 0,C 180,E1 35261.103,E2 35261.103} C_VEL
LIN {X 0,Y 739.127,Z 649.029,A -85,B 0,C 180,E1 35260.89,E2 35260.89} C_VEL
LIN {X 0,Y 736.081,Z 640.979,A -85,B 0,C 180,E1 35260.047,E2 35260.047} C_VEL
LIN {X 0,Y 736.075,Z 640.975,A -85,B 0,C 180,E1 35257.223,E2 35257.223} C_VEL
LIN {X 0,Y 736.088,Z 640.981,A -85,B 0,C 180,E1 35254.321,E2 35254.321} C_VEL
LIN {X 0,Y 736.098,Z 640.969,A -85,B 0,C 180,E1 35251.339,E2 35251.339} C_VEL
LIN {X 0,Y 736.096,Z 640.982,A -85,B 0,C 180,E1 35248.245,E2 35248.245} C_VEL
LIN {X 0,Y 736.093,Z 640.97,A -85,B 0,C 180,E1 35245.213,E2 35245.213} C_VEL
LIN {X 0,Y 736.09,Z 640.982,A -85,B 0,C 180,E1 35242.22,E2 35242.22} C_VEL
LIN {X 0,Y 736.074,Z 640.974,A -85,B 0,C 180,E1 35239.304,E2 35239.304} C_VEL
LIN {X 0,Y 736.08,Z 640.975,A -85,B 0,C 180,E1 35236.472,E2 35236.472} C_VEL
LIN {X 0,Y 736.087,Z 640.981,A -85,B 0,C 180,E1 35233.525,E2 35233.525} C_VEL
LIN {X 0,Y 736.109,Z 641.187,A -85,B 0,C 180,E1 35232.109,E2 35232.109} C_VEL
LIN {X 0,Y 738.825,Z 648.354,A -85,B 0,C 180,E1 35231.584,E2 35231.584} C_VEL
LIN {X 0,Y 738.193,Z 699.743,A -85,B 0,C 180,E1 35229.037,E2 35229.037} C_VEL
LIN {X 0,Y 738.338,Z 753.231,A -85,B 0,C 180,E1 35226.476,E2 35226.476} C_VEL
LIN {X 0,Y 740.198,Z 769.259,A -85,B 0,C 180,E1 35225.656,E2 35225.656} C_VEL
LIN {X 0,Y 743.119,Z 779.693,A -85,B 0,C 180,E1 35225.066,E2 35225.066} C_VEL
LIN {X 0,Y 746.038,Z 785.708,A -85,B 0,C 180,E1 35224.621,E2 35224.621} C_VEL
LIN {X 0,Y 748.576,Z 789.088,A -85,B 0,C 180,E1 35224.216,E2 35224.216} C_VEL
LIN {X 0,Y 750.816,Z 790.849,A -85,B 0,C 180,E1 35223.797,E2 35223.797} C_VEL
LIN {X 0,Y 752.668,Z 791.034,A -85,B 0,C 180,E1 35223.321,E2 35223.321} C_VEL
LIN {X 0,Y 753.527,Z 789.528,A -85,B 0,C 180,E1 35222.864,E2 35222.864} C_VEL
LIN {X 0,Y 753.28,Z 786.484,A -85,B 0,C 180,E1 35222.45,E2 35222.45} C_VEL
LIN {X 0,Y 751.951,Z 782.114,A -85,B 0,C 180,E1 35222.111,E2 35222.111} C_VEL
LIN {X 0,Y 749.628,Z 775.314,A -85,B 0,C 180,E1 35221.815,E2 35221.815} C_VEL
LIN {X 0,Y 748.002,Z 766.927,A -85,B 0,C 180,E1 35221.614,E2 35221.614} C_VEL
LIN {X 0,Y 747.18,Z 756.52,A -85,B 0,C 180,E1 35221.511,E2 35221.511} C_VEL
LIN {X 0,Y 747.069,Z 655.532,A -85,B 0,C 180,E1 35221.497,E2 35221.497} C_VEL
LIN {X 0,Y 743.244,Z 665.044,A -85,B 0,C 180,E1 35221.012,E2 35221.012} C_VEL
LIN {X 0,Y 740.552,Z 669.578,A -85,B 0,C 180,E1 35220.664,E2 35220.664} C_VEL
LIN {X 0,Y 739.154,Z 670.68,A -85,B 0,C 180,E1 35220.481,E2 35220.481} C_VEL
LIN {X 0,Y 738.345,Z 670.472,A -85,B 0,C 180,E1 35220.372,E2 35220.372} C_VEL
LIN {X 0,Y 737.912,Z 729.219,A -85,B 0,C 180,E1 35217.519,E2 35217.519} C_VEL
LIN {X 0,Y 737.802,Z 757.956,A -85,B 0,C 180,E1 35216.168,E2 35216.168} C_VEL
LIN {X 0,Y 738.229,Z 763.831,A -85,B 0,C 180,E1 35216.089,E2 35216.089} C_VEL
LIN {X 0,Y 737.783,Z 1030.896,A -85,B 0,C 180,E1 35213.303,E2 35213.303} C_VEL
LIN {X 0,Y 737.682,Z 1066.305,A -85,B 0,C 180,E1 35212.905,E2 35212.905} C_VEL
LIN {X 0,Y 737.592,Z 1088.45,A -85,B 0,C 180,E1 35212.505,E2 35212.505} C_VEL
LIN {X 0,Y 737.424,Z 1109.775,A -85,B 0,C 180,E1 35211.975,E2 35211.975} C_VEL
LIN {X 0,Y 737.26,Z 1130.72,A -85,B 0,C 180,E1 35211.312,E2 35211.312} C_VEL
LIN {X 0,Y 737.102,Z 1150.763,A -85,B 0,C 180,E1 35210.526,E2 35210.526} C_VEL
LIN {X 0,Y 736.892,Z 1170.772,A -85,B 0,C 180,E1 35209.58,E2 35209.58} C_VEL
LIN {X 0,Y 736.683,Z 1190.481,A -85,B 0,C 180,E1 35208.476,E2 35208.476} C_VEL
LIN {X 0,Y 736.522,Z 1208.393,A -85,B 0,C 180,E1 35207.295,E2 35207.295} C_VEL
LIN {X 0,Y 736.373,Z 1225.487,A -85,B 0,C 180,E1 35205.978,E2 35205.978} C_VEL
LIN {X 0,Y 736.231,Z 1240.433,A -85,B 0,C 180,E1 35204.631,E2 35204.631} C_VEL
LIN {X 0,Y 736.114,Z 1254.176,A -85,B 0,C 180,E1 35203.19,E2 35203.19} C_VEL
LIN {X 0,Y 736.04,Z 1266.83,A -85,B 0,C 180,E1 35201.632,E2 35201.632} C_VEL
LIN {X 0,Y 735.98,Z 1276.884,A -85,B 0,C 180,E1 35200.171,E2 35200.171} C_VEL
LIN {X 0,Y 735.942,Z 1285.898,A -85,B 0,C 180,E1 35198.594,E2 35198.594} C_VEL
LIN {X 0,Y 735.92,Z 1293.555,A -85,B 0,C 180,E1 35196.944,E2 35196.944} C_VEL
LIN {X 0,Y 735.921,Z 1299.156,A -85,B 0,C 180,E1 35195.378,E2 35195.378} C_VEL
LIN {X 0,Y 735.913,Z 1303.635,A -85,B 0,C 180,E1 35193.66,E2 35193.66} C_VEL
LIN {X 0,Y 735.912,Z 1306.407,A -85,B 0,C 180,E1 35191.945,E2 35191.945} C_VEL
LIN {X 0,Y 735.899,Z 1307.418,A -85,B 0,C 180,E1 35190.31,E2 35190.31} C_VEL
LIN {X 0,Y 735.905,Z 1306.822,A -85,B 0,C 180,E1 35188.52,E2 35188.52} C_VEL
LIN {X 0,Y 735.918,Z 1304.576,A -85,B 0,C 180,E1 35186.806,E2 35186.806} C_VEL
LIN {X 0,Y 735.908,Z 1300.58,A -85,B 0,C 180,E1 35185.089,E2 35185.089} C_VEL
LIN {X 0,Y 735.914,Z 1295.065,A -85,B 0,C 180,E1 35183.446,E2 35183.446} C_VEL
LIN {X 0,Y 735.949,Z 1287.918,A -85,B 0,C 180,E1 35181.797,E2 35181.797} C_VEL
LIN {X 0,Y 735.977,Z 1278.835,A -85,B 0,C 180,E1 35180.143,E2 35180.143} C_VEL
LIN {X 0,Y 736.032,Z 1268.794,A -85,B 0,C 180,E1 35178.639,E2 35178.639} C_VEL
LIN {X 0,Y 736.108,Z 1257.662,A -85,B 0,C 180,E1 35177.207,E2 35177.207} C_VEL
LIN {X 0,Y 736.209,Z 1243.686,A -85,B 0,C 180,E1 35175.688,E2 35175.688} C_VEL
LIN {X 0,Y 736.322,Z 1228.928,A -85,B 0,C 180,E1 35174.321,E2 35174.321} C_VEL
LIN {X 0,Y 736.476,Z 1212.238,A -85,B 0,C 180,E1 35172.987,E2 35172.987} C_VEL
LIN {X 0,Y 736.666,Z 1194.411,A -85,B 0,C 180,E1 35171.767,E2 35171.767} C_VEL
LIN {X 0,Y 736.86,Z 1175.503,A -85,B 0,C 180,E1 35170.664,E2 35170.664} C_VEL
LIN {X 0,Y 737.04,Z 1155.395,A -85,B 0,C 180,E1 35169.677,E2 35169.677} C_VEL
LIN {X 0,Y 737.216,Z 1135.139,A -85,B 0,C 180,E1 35168.851,E2 35168.851} C_VEL
LIN {X 0,Y 737.411,Z 1114.104,A -85,B 0,C 180,E1 35168.147,E2 35168.147} C_VEL
LIN {X 0,Y 737.552,Z 1092.538,A -85,B 0,C 180,E1 35167.584,E2 35167.584} C_VEL
LIN {X 0,Y 737.67,Z 1070.721,A -85,B 0,C 180,E1 35167.165,E2 35167.165} C_VEL
LIN {X 0,Y 737.759,Z 1045.981,A -85,B 0,C 180,E1 35166.853,E2 35166.853} C_VEL
LIN {X 0,Y 738.214,Z 775.597,A -85,B 0,C 180,E1 35164.035,E2 35164.035} C_VEL
LIN {X 0,Y 737.992,Z 759.164,A -85,B 0,C 180,E1 35163.852,E2 35163.852} C_VEL
LIN {X 0,Y 737.715,Z 756.909,A -85,B 0,C 180,E1 35163.802,E2 35163.802} C_VEL
LIN {X 0,Y 738.115,Z 699.734,A -85,B 0,C 180,E1 35161.058,E2 35161.058} C_VEL
LIN {X 0,Y 738.408,Z 670.485,A -85,B 0,C 180,E1 35159.617,E2 35159.617} C_VEL
LIN {X 0,Y 739.676,Z 670.427,A -85,B 0,C 180,E1 35159.45,E2 35159.45} C_VEL
LIN {X 0,Y 741.972,Z 667.469,A -85,B 0,C 180,E1 35159.151,E2 35159.151} C_VEL
LIN {X 0,Y 745.521,Z 659.755,A -85,B 0,C 180,E1 35158.698,E2 35158.698} C_VEL
LIN {X 0,Y 747.094,Z 655.462,A -85,B 0,C 180,E1 35158.5,E2 35158.5} C_VEL
LIN {X 0,Y 747.231,Z 757.857,A -85,B 0,C 180,E1 35158.483,E2 35158.483} C_VEL
LIN {X 0,Y 748.147,Z 768.008,A -85,B 0,C 180,E1 35158.368,E2 35158.368} C_VEL
LIN {X 0,Y 749.84,Z 776.085,A -85,B 0,C 180,E1 35158.159,E2 35158.159} C_VEL
LIN {X 0,Y 752.16,Z 782.697,A -85,B 0,C 180,E1 35157.854,E2 35157.854} C_VEL
LIN {X 0,Y 753.363,Z 786.903,A -85,B 0,C 180,E1 35157.506,E2 35157.506} C_VEL
LIN {X 0,Y 753.478,Z 789.802,A -85,B 0,C 180,E1 35157.083,E2 35157.083} C_VEL
LIN {X 0,Y 752.501,Z 791.109,A -85,B 0,C 180,E1 35156.625,E2 35156.625} C_VEL
LIN {X 0,Y 750.636,Z 790.749,A -85,B 0,C 180,E1 35156.165,E2 35156.165} C_VEL
LIN {X 0,Y 748.536,Z 789.05,A -85,B 0,C 180,E1 35155.778,E2 35155.778} C_VEL
LIN {X 0,Y 745.943,Z 785.55,A -85,B 0,C 180,E1 35155.364,E2 35155.364} C_VEL
LIN {X 0,Y 742.791,Z 778.715,A -85,B 0,C 180,E1 35154.863,E2 35154.863} C_VEL
LIN {X 0,Y 740.196,Z 767.796,A -85,B 0,C 180,E1 35154.202,E2 35154.202} C_VEL
LIN {X 0,Y 738.818,Z 751.229,A -85,B 0,C 180,E1 35153.308,E2 35153.308} C_VEL
LIN {X 0,Y 739.205,Z 693.254,A -85,B 0,C 180,E1 35150.323,E2 35150.323} C_VEL
LIN {X 0,Y 739.642,Z 649.649,A -85,B 0,C 180,E1 35147.997,E2 35147.997} C_VEL
LIN {X 0,Y 736.179,Z 641.512,A -85,B 0,C 180,E1 35147.331,E2 35147.331} C_VEL
LIN {X 0,Y 736.092,Z 640.983,A -85,B 0,C 180,E1 35147.278,E2 35147.278} C_VEL
LIN {X 0,Y 736.097,Z 640.977,A -85,B 0,C 180,E1 35144.283,E2 35144.283} C_VEL
LIN {X 0,Y 736.092,Z 640.978,A -85,B 0,C 180,E1 35141.21,E2 35141.21} C_VEL
LIN {X 0,Y 736.094,Z 640.981,A -85,B 0,C 180,E1 35138.266,E2 35138.266} C_VEL
LIN {X 0,Y 736.096,Z 640.981,A -85,B 0,C 180,E1 35135.357,E2 35135.357} C_VEL
LIN {X 0,Y 736.077,Z 640.981,A -85,B 0,C 180,E1 35132.451,E2 35132.451} C_VEL
LIN {X 0,Y 736.11,Z 641.088,A -85,B 0,C 180,E1 35130.736,E2 35130.736} C_VEL
LIN {X 0,Y 737.679,Z 647.093,A -85,B 0,C 180,E1 35130.19,E2 35130.19} C_VEL
LIN {X 0,Y 737.355,Z 684.851,A -85,B 0,C 180,E1 35127.281,E2 35127.281} C_VEL
LIN {X 0,Y 737.318,Z 700.558,A -85,B 0,C 180,E1 35126.114,E2 35126.114} C_VEL
LIN {X 0,Y 738.23,Z 705.807,A -85,B 0,C 180,E1 35126.023,E2 35126.023} C_VEL
LIN {X 0,Y 737.757,Z 989.076,A -85,B 0,C 180,E1 35123.07,E2 35123.07} C_VEL
LIN {X 0,Y 737.667,Z 1012.557,A -85,B 0,C 180,E1 35122.759,E2 35122.759} C_VEL
LIN {X 0,Y 737.526,Z 1035.225,A -85,B 0,C 180,E1 35122.307,E2 35122.307} C_VEL
LIN {X 0,Y 737.395,Z 1056.238,A -85,B 0,C 180,E1 35121.744,E2 35121.744} C_VEL
LIN {X 0,Y 737.206,Z 1077.292,A -85,B 0,C 180,E1 35121.023,E2 35121.023} C_VEL
LIN {X 0,Y 737.006,Z 1098.276,A -85,B 0,C 180,E1 35120.143,E2 35120.143} C_VEL
LIN {X 0,Y 736.828,Z 1117.508,A -85,B 0,C 180,E1 35119.181,E2 35119.181} C_VEL
LIN {X 0,Y 736.652,Z 1135.649,A -85,B 0,C 180,E1 35118.109,E2 35118.109} C_VEL
LIN {X 0,Y 736.471,Z 1152.723,A -85,B 0,C 180,E1 35116.931,E2 35116.931} C_VEL
LIN {X 0,Y 736.316,Z 1169.359,A -85,B 0,C 180,E1 35115.598,E2 35115.598} C_VEL
LIN {X 0,Y 736.202,Z 1184.024,A -85,B 0,C 180,E1 35114.231,E2 35114.231} C_VEL
LIN {X 0,Y 736.109,Z 1197.529,A -85,B 0,C 180,E1 35112.763,E2 35112.763} C_VEL
LIN {X 0,Y 736.027,Z 1209.401,A -85,B 0,C 180,E1 35111.235,E2 35111.235} C_VEL
LIN {X 0,Y 735.974,Z 1219.951,A -85,B 0,C 180,E1 35109.62,E2 35109.62} C_VEL
LIN {X 0,Y 735.946,Z 1228.481,A -85,B 0,C 180,E1 35108.044,E2 35108.044} C_VEL
LIN {X 0,Y 735.92,Z 1235.497,A -85,B 0,C 180,E1 35106.397,E2 35106.397} C_VEL
LIN {X 0,Y 735.915,Z 1241.075,A -85,B 0,C 180,E1 35104.676,E2 35104.676} C_VEL
LIN {X 0,Y 735.898,Z 1244.792,A -85,B 0,C 180,E1 35103.038,E2 35103.038} C_VEL
LIN {X 0,Y 735.906,Z 1246.909,A -85,B 0,C 180,E1 35101.324,E2 35101.324} C_VEL
LIN {X 0,Y 735.917,Z 1247.386,A -85,B 0,C 180,E1 35099.533,E2 35099.533} C_VEL
LIN {X 0,Y 735.902,Z 1246.183,A -85,B 0,C 180,E1 35097.82,E2 35097.82} C_VEL
LIN {X 0,Y 735.901,Z 1243.241,A -85,B 0,C 180,E1 35096.105,E2 35096.105} C_VEL
LIN {X 0,Y 735.918,Z 1238.797,A -85,B 0,C 180,E1 35094.464,E2 35094.464} C_VEL
LIN {X 0,Y 735.935,Z 1232.785,A -85,B 0,C 180,E1 35092.819,E2 35092.819} C_VEL
LIN {X 0,Y 735.949,Z 1225.3,A -85,B 0,C 180,E1 35091.247,E2 35091.247} C_VEL
LIN {X 0,Y 735.991,Z 1215.62,A -85,B 0,C 180,E1 35089.59,E2 35089.59} C_VEL
LIN {X 0,Y 735.996,Z 1214.931,A -85,B 0,C 180,E1 35089.485,E2 35089.485} C_VEL
LIN {X 0,Y 735.027,Z 1211.496,A -85,B 0,C 180,E1 35088.95,E2 35088.95} C_VEL
LIN {X 0,Y 728.862,Z 1201.795,A -85,B 0,C 180,E1 35087.546,E2 35087.546} C_VEL
LIN {X 0,Y 728.169,Z 1198.333,A -85,B 0,C 180,E1 35087.101,E2 35087.101} C_VEL
LIN {X 0,Y 728.296,Z 1184.889,A -85,B 0,C 180,E1 35085.611,E2 35085.611} C_VEL
LIN {X 0,Y 728.455,Z 1170.021,A -85,B 0,C 180,E1 35084.198,E2 35084.198} C_VEL
LIN {X 0,Y 728.665,Z 1153.384,A -85,B 0,C 180,E1 35082.841,E2 35082.841} C_VEL
LIN {X 0,Y 728.906,Z 1136.767,A -85,B 0,C 180,E1 35081.671,E2 35081.671} C_VEL
LIN {X 0,Y 729.132,Z 1118.513,A -85,B 0,C 180,E1 35080.576,E2 35080.576} C_VEL
LIN {X 0,Y 729.384,Z 1098.928,A -85,B 0,C 180,E1 35079.577,E2 35079.577} C_VEL
LIN {X 0,Y 729.651,Z 1078.56,A -85,B 0,C 180,E1 35078.706,E2 35078.706} C_VEL
LIN {X 0,Y 729.889,Z 1058.077,A -85,B 0,C 180,E1 35077.989,E2 35077.989} C_VEL
LIN {X 0,Y 730.087,Z 1036.648,A -85,B 0,C 180,E1 35077.398,E2 35077.398} C_VEL
LIN {X 0,Y 730.268,Z 1013.948,A -85,B 0,C 180,E1 35076.929,E2 35076.929} C_VEL
LIN {X 0,Y 730.389,Z 991.216,A -85,B 0,C 180,E1 35076.615,E2 35076.615} C_VEL
LIN {X 0,Y 731.037,Z 705.962,A -85,B 0,C 180,E1 35073.612,E2 35073.612} C_VEL
LIN {X 0,Y 729.728,Z 699.886,A -85,B 0,C 180,E1 35073.478,E2 35073.478} C_VEL
LIN {X 0,Y 730.13,Z 661.974,A -85,B 0,C 180,E1 35070.551,E2 35070.551} C_VEL
LIN {X 0,Y 730.048,Z 648.54,A -85,B 0,C 180,E1 35069.485,E2 35069.485} C_VEL
LIN {X 0,Y 728.139,Z 641.968,A -85,B 0,C 180,E1 35068.868,E2 35068.868} C_VEL
LIN {X 0,Y 728.159,Z 641.967,A -85,B 0,C 180,E1 35066.021,E2 35066.021} C_VEL
LIN {X 0,Y 728.156,Z 641.962,A -85,B 0,C 180,E1 35063.026,E2 35063.026} C_VEL
LIN {X 0,Y 728.163,Z 641.965,A -85,B 0,C 180,E1 35060.011,E2 35060.011} C_VEL
LIN {X 0,Y 728.144,Z 641.968,A -85,B 0,C 180,E1 35057.048,E2 35057.048} C_VEL
LIN {X 0,Y 728.134,Z 641.964,A -85,B 0,C 180,E1 35054.207,E2 35054.207} C_VEL
LIN {X 0,Y 728.141,Z 641.971,A -85,B 0,C 180,E1 35051.31,E2 35051.31} C_VEL
LIN {X 0,Y 728.151,Z 641.964,A -85,B 0,C 180,E1 35048.363,E2 35048.363} C_VEL
LIN {X 0,Y 728.158,Z 641.961,A -85,B 0,C 180,E1 35045.318,E2 35045.318} C_VEL
LIN {X 0,Y 728.157,Z 641.965,A -85,B 0,C 180,E1 35042.233,E2 35042.233} C_VEL
LIN {X 0,Y 728.149,Z 641.966,A -85,B 0,C 180,E1 35039.266,E2 35039.266} C_VEL
LIN {X 0,Y 728.14,Z 641.962,A -85,B 0,C 180,E1 35036.331,E2 35036.331} C_VEL
LIN {X 0,Y 728.155,Z 641.968,A -85,B 0,C 180,E1 35033.467,E2 35033.467} C_VEL
LIN {X 0,Y 728.151,Z 641.964,A -85,B 0,C 180,E1 35030.498,E2 35030.498} C_VEL
LIN {X 0,Y 728.153,Z 641.961,A -85,B 0,C 180,E1 35027.585,E2 35027.585} C_VEL
LIN {X 0,Y 728.157,Z 641.966,A -85,B 0,C 180,E1 35024.512,E2 35024.512} C_VEL
LIN {X 0,Y 728.152,Z 641.964,A -85,B 0,C 180,E1 35021.566,E2 35021.566} C_VEL
LIN {X 0,Y 728.141,Z 641.961,A -85,B 0,C 180,E1 35018.609,E2 35018.609} C_VEL
LIN {X 0,Y 728.151,Z 641.97,A -85,B 0,C 180,E1 35015.754,E2 35015.754} C_VEL
LIN {X 0,Y 728.14,Z 641.963,A -85,B 0,C 180,E1 35012.835,E2 35012.835} C_VEL
LIN {X 0,Y 728.156,Z 641.961,A -85,B 0,C 180,E1 35009.922,E2 35009.922} C_VEL
LIN {X 0,Y 728.157,Z 641.971,A -85,B 0,C 180,E1 35006.931,E2 35006.931} C_VEL
LIN {X 0,Y 728.148,Z 641.963,A -85,B 0,C 180,E1 35003.932,E2 35003.932} C_VEL
LIN {X 0,Y 728.137,Z 641.964,A -85,B 0,C 180,E1 35000.995,E2 35000.995} C_VEL
LIN {X 0,Y 728.148,Z 641.969,A -85,B 0,C 180,E1 34998.114,E2 34998.114} C_VEL
LIN {X 0,Y 728.144,Z 641.962,A -85,B 0,C 180,E1 34995.181,E2 34995.181} C_VEL
LIN {X 0,Y 728.156,Z 641.964,A -85,B 0,C 180,E1 34992.253,E2 34992.253} C_VEL
LIN {X 0,Y 728.156,Z 641.968,A -85,B 0,C 180,E1 34989.251,E2 34989.251} C_VEL
LIN {X 0,Y 728.144,Z 641.963,A -85,B 0,C 180,E1 34986.277,E2 34986.277} C_VEL
LIN {X 0,Y 728.147,Z 641.965,A -85,B 0,C 180,E1 34983.375,E2 34983.375} C_VEL
LIN {X 0,Y 728.153,Z 641.966,A -85,B 0,C 180,E1 34980.466,E2 34980.466} C_VEL
LIN {X 0,Y 728.145,Z 641.96,A -85,B 0,C 180,E1 34977.528,E2 34977.528} C_VEL
LIN {X 0,Y 728.153,Z 641.964,A -85,B 0,C 180,E1 34974.519,E2 34974.519} C_VEL
LIN {X 0,Y 728.161,Z 641.967,A -85,B 0,C 180,E1 34971.536,E2 34971.536} C_VEL
LIN {X 0,Y 728.157,Z 641.961,A -85,B 0,C 180,E1 34968.451,E2 34968.451} C_VEL
LIN {X 0,Y 728.148,Z 641.965,A -85,B 0,C 180,E1 34965.439,E2 34965.439} C_VEL
LIN {X 0,Y 728.143,Z 641.972,A -85,B 0,C 180,E1 34962.491,E2 34962.491} C_VEL
LIN {X 0,Y 728.138,Z 641.968,A -85,B 0,C 180,E1 34959.684,E2 34959.684} C_VEL
LIN {X 0,Y 728.151,Z 642.081,A -85,B 0,C 180,E1 34959.414,E2 34959.414} C_VEL
LIN {X 0,Y 730.808,Z 650.456,A -85,B 0,C 180,E1 34958.702,E2 34958.702} C_VEL
LIN {X 0,Y 730.4,Z 695.159,A -85,B 0,C 180,E1 34955.675,E2 34955.675} C_VEL
LIN {X 0,Y 729.685,Z 738.667,A -85,B 0,C 180,E1 34952.77,E2 34952.77} C_VEL
LIN {X 0,Y 729.13,Z 782.662,A -85,B 0,C 180,E1 34949.9,E2 34949.9} C_VEL
LIN {X 0,Y 728.78,Z 825.462,A -85,B 0,C 180,E1 34947.186,E2 34947.186} C_VEL
LIN {X 0,Y 728.501,Z 872.368,A -85,B 0,C 180,E1 34944.277,E2 34944.277} C_VEL
LIN {X 0,Y 728.468,Z 891.745,A -85,B 0,C 180,E1 34943.109,E2 34943.109} C_VEL
LIN {X 0,Y 728.526,Z 1032.743,A -85,B 0,C 180,E1 34941.693,E2 34941.693} C_VEL
LIN {X 0,Y 728.474,Z 1047.889,A -85,B 0,C 180,E1 34941.42,E2 34941.42} C_VEL
LIN {X 0,Y 728.397,Z 1064.358,A -85,B 0,C 180,E1 34940.967,E2 34940.967} C_VEL
LIN {X 0,Y 728.293,Z 1078.907,A -85,B 0,C 180,E1 34940.409,E2 34940.409} C_VEL
LIN {X 0,Y 728.209,Z 1091.758,A -85,B 0,C 180,E1 34939.781,E2 34939.781} C_VEL
LIN {X 0,Y 728.148,Z 1103.451,A -85,B 0,C 180,E1 34939.076,E2 34939.076} C_VEL
LIN {X 0,Y 728.083,Z 1114.208,A -85,B 0,C 180,E1 34938.289,E2 34938.289} C_VEL
LIN {X 0,Y 728.023,Z 1124.861,A -85,B 0,C 180,E1 34937.34,E2 34937.34} C_VEL
LIN {X 0,Y 727.97,Z 1135.036,A -85,B 0,C 180,E1 34936.19,E2 34936.19} C_VEL
LIN {X 0,Y 727.943,Z 1142.699,A -85,B 0,C 180,E1 34935.073,E2 34935.073} C_VEL
LIN {X 0,Y 727.924,Z 1148.451,A -85,B 0,C 180,E1 34933.99,E2 34933.99} C_VEL
LIN {X 0,Y 727.917,Z 1153.137,A -85,B 0,C 180,E1 34932.776,E2 34932.776} C_VEL
LIN {X 0,Y 727.916,Z 1156.344,A -85,B 0,C 180,E1 34931.409,E2 34931.409} C_VEL
LIN {X 0,Y 727.916,Z 1157.445,A -85,B 0,C 180,E1 34930.127,E2 34930.127} C_VEL
LIN {X 0,Y 727.916,Z 1156.879,A -85,B 0,C 180,E1 34928.93,E2 34928.93} C_VEL
LIN {X 0,Y 727.918,Z 1154.794,A -85,B 0,C 180,E1 34927.736,E2 34927.736} C_VEL
LIN {X 0,Y 727.924,Z 1150.815,A -85,B 0,C 180,E1 34926.467,E2 34926.467} C_VEL
LIN {X 0,Y 727.934,Z 1144.848,A -85,B 0,C 180,E1 34925.201,E2 34925.201} C_VEL
LIN {X 0,Y 727.956,Z 1137.802,A -85,B 0,C 180,E1 34924.096,E2 34924.096} C_VEL
LIN {X 0,Y 727.99,Z 1129.53,A -85,B 0,C 180,E1 34923.071,E2 34923.071} C_VEL
LIN {X 0,Y 728.048,Z 1120.12,A -85,B 0,C 180,E1 34922.125,E2 34922.125} C_VEL
LIN {X 0,Y 728.13,Z 1107.44,A -85,B 0,C 180,E1 34921.102,E2 34921.102} C_VEL
LIN {X 0,Y 728.211,Z 1094.408,A -85,B 0,C 180,E1 34920.275,E2 34920.275} C_VEL
LIN {X 0,Y 728.262,Z 1082.118,A -85,B 0,C 180,E1 34919.646,E2 34919.646} C_VEL
LIN {X 0,Y 728.365,Z 1069.702,A -85,B 0,C 180,E1 34919.135,E2 34919.135} C_VEL
LIN {X 0,Y 728.437,Z 1056.238,A -85,B 0,C 180,E1 34918.702,E2 34918.702} C_VEL
LIN {X 0,Y 728.497,Z 1040.645,A -85,B 0,C 180,E1 34918.341,E2 34918.341} C_VEL
LIN {X 0,Y 728.558,Z 1021.22,A -85,B 0,C 180,E1 34918.083,E2 34918.083} C_VEL
LIN {X 0,Y 728.468,Z 891.781,A -85,B 0,C 180,E1 34916.801,E2 34916.801} C_VEL
LIN {X 0,Y 728.431,Z 886.422,A -85,B 0,C 180,E1 34916.498,E2 34916.498} C_VEL
LIN {X 0,Y 728.701,Z 839.815,A -85,B 0,C 180,E1 34913.619,E2 34913.619} C_VEL
LIN {X 0,Y 729.049,Z 793.917,A -85,B 0,C 180,E1 34910.726,E2 34910.726} C_VEL
LIN {X 0,Y 730.172,Z 750.215,A -85,B 0,C 180,E1 34907.745,E2 34907.745} C_VEL
LIN {X 0,Y 731.564,Z 708.405,A -85,B 0,C 180,E1 34904.827,E2 34904.827} C_VEL
LIN {X 0,Y 732.141,Z 685.841,A -85,B 0,C 180,E1 34903.201,E2 34903.201} C_VEL
LIN {X 0,Y 732.675,Z 653.617,A -85,B 0,C 180,E1 34900.795,E2 34900.795} C_VEL
LIN {X 0,Y 728.149,Z 641.967,A -85,B 0,C 180,E1 34899.544,E2 34899.544} C_VEL
LIN {X 0,Y 728.158,Z 641.97,A -85,B 0,C 180,E1 34896.527,E2 34896.527} C_VEL
LIN {X 0,Y 728.157,Z 641.959,A -85,B 0,C 180,E1 34893.494,E2 34893.494} C_VEL
LIN {X 0,Y 728.161,Z 641.97,A -85,B 0,C 180,E1 34890.373,E2 34890.373} C_VEL
LIN {X 0,Y 728.159,Z 641.959,A -85,B 0,C 180,E1 34887.246,E2 34887.246} C_VEL
LIN {X 0,Y 728.154,Z 641.971,A -85,B 0,C 180,E1 34884.198,E2 34884.198} C_VEL
LIN {X 0,Y 728.143,Z 641.961,A -85,B 0,C 180,E1 34881.231,E2 34881.231} C_VEL
LIN {X 0,Y 728.141,Z 641.967,A -85,B 0,C 180,E1 34878.331,E2 34878.331} C_VEL
LIN {X 0,Y 728.139,Z 641.968,A -85,B 0,C 180,E1 34875.435,E2 34875.435} C_VEL
LIN {X 0,Y 728.172,Z 642.112,A -85,B 0,C 180,E1 34872.52,E2 34872.52} C_VEL
LIN {X 0,Y 731.889,Z 651.527,A -85,B 0,C 180,E1 34871.796,E2 34871.796} C_VEL
LIN {X 0,Y 731.011,Z 701.645,A -85,B 0,C 180,E1 34869.268,E2 34869.268} C_VEL
LIN {X 0,Y 730.936,Z 754.347,A -85,B 0,C 180,E1 34866.71,E2 34866.71} C_VEL
LIN {X 0,Y 732.819,Z 771.502,A -85,B 0,C 180,E1 34865.825,E2 34865.825} C_VEL
LIN {X 0,Y 735.619,Z 782.132,A -85,B 0,C 180,E1 34865.223,E2 34865.223} C_VEL
LIN {X 0,Y 739.765,Z 790.61,A -85,B 0,C 180,E1 34864.681,E2 34864.681} C_VEL
LIN {X 0,Y 743.169,Z 794.908,A -85,B 0,C 180,E1 34864.299,E2 34864.299} C_VEL
LIN {X 0,Y 746.524,Z 797.615,A -85,B 0,C 180,E1 34863.857,E2 34863.857} C_VEL
LIN {X 0,Y 748.951,Z 798.502,A -85,B 0,C 180,E1 34863.445,E2 34863.445} C_VEL
LIN {X 0,Y 750.814,Z 797.951,A -85,B 0,C 180,E1 34862.965,E2 34862.965} C_VEL
LIN {X 0,Y 751.493,Z 795.932,A -85,B 0,C 180,E1 34862.514,E2 34862.514} C_VEL
LIN {X 0,Y 750.949,Z 792.647,A -85,B 0,C 180,E1 34862.104,E2 34862.104} C_VEL
LIN {X 0,Y 749.23,Z 788.239,A -85,B 0,C 180,E1 34861.766,E2 34861.766} C_VEL
LIN {X 0,Y 746.417,Z 780.789,A -85,B 0,C 180,E1 34861.415,E2 34861.415} C_VEL
LIN {X 0,Y 744.438,Z 772.085,A -85,B 0,C 180,E1 34861.165,E2 34861.165} C_VEL
LIN {X 0,Y 743.26,Z 761.612,A -85,B 0,C 180,E1 34861.015,E2 34861.015} C_VEL
LIN {X 0,Y 742.952,Z 751.201,A -85,B 0,C 180,E1 34860.975,E2 34860.975} C_VEL
LIN {X 0,Y 742.857,Z 676.201,A -85,B 0,C 180,E1 34860.963,E2 34860.963} C_VEL
